C01812=1216.851,306.923,-68.303,-176.403,7.071,148.270
C01813=1216.855,306.675,-68.273,-176.405,7.069,148.270
C01814=1216.859,306.427,-68.243,-176.408,7.066,148.270
C01815=1216.864,306.178,-68.213,-176.410,7.063,148.270
C01816=1216.868,305.930,-68.183,-176.413,7.060,148.270
C01817=1216.872,305.682,-68.154,-176.415,7.058,148.270
C01818=1216.876,305.434,-68.124,-176.417,7.056,148.270
C01819=1216.881,305.186,-68.095,-176.420,7.053,148.270
C01820=1216.885,304.938,-68.064,-176.422,7.051,148.270
C01821=1216.889,304.690,-68.035,-176.424,7.048,148.270
C01822=1216.894,304.442,-68.006,-176.427,7.045,148.270
C01823=1216.898,304.193,-67.976,-176.429,7.042,148.270
C01824=1216.903,303.945,-67.946,-176.431,7.040,148.270
C01825=1216.907,303.697,-67.916,-176.434,7.038,148.270
C01826=1216.911,303.449,-67.886,-176.436,7.035,148.270
C01827=1216.915,303.201,-67.857,-176.438,7.033,148.270
C01828=1216.919,302.952,-67.827,-176.441,7.030,148.270
C01829=1216.924,302.704,-67.797,-176.443,7.028,148.270
C01830=1216.928,302.456,-67.768,-176.446,7.024,148.270
C01831=1216.932,302.207,-67.739,-176.448,7.022,148.270
C01832=1216.936,301.960,-67.708,-176.451,7.019,148.270
C01833=1216.940,301.711,-67.679,-176.453,7.017,148.270
C01834=1216.945,301.463,-67.649,-176.455,7.015,148.270
C01835=1216.950,301.215,-67.619,-176.457,7.012,148.271
C01836=1216.954,300.966,-67.590,-176.460,7.010,148.271
C01837=1216.958,300.718,-67.561,-176.463,7.007,148.271
C01838=1216.963,300.470,-67.531,-176.465,7.005,148.271
C01839=1216.967,300.222,-67.502,-176.468,7.002,148.271
C01840=1216.971,299.974,-67.473,-176.470,6.999,148.271
C01841=1216.975,299.726,-67.443,-176.472,6.997,148.271
C01842=1216.979,299.477,-67.414,-176.474,6.994,148.271
C01843=1216.984,299.229,-67.384,-176.477,6.992,148.271
C01844=1216.988,298.981,-67.355,-176.479,6.989,148.271
C01845=1216.992,298.733,-67.325,-176.481,6.987,148.271
C01846=1216.996,298.484,-67.296,-176.484,6.985,148.271
C01847=1217.001,298.237,-67.267,-176.487,6.982,148.271
C01848=1217.005,297.988,-67.238,-176.489,6.980,148.271
C01849=1217.010,297.740,-67.209,-176.491,6.976,148.271
C01850=1217.014,297.491,-67.179,-176.493,6.974,148.272
C01851=1217.018,297.243,-67.150,-176.496,6.971,148.272
C01852=1217.022,296.995,-67.120,-176.498,6.969,148.272
C01853=1217.026,296.747,-67.091,-176.500,6.967,148.272
C01854=1217.031,296.499,-67.062,-176.504,6.964,148.272
C01855=1217.036,296.250,-67.033,-176.506,6.962,148.272
C01856=1217.040,296.002,-67.003,-176.508,6.959,148.272
C01857=1217.044,295.754,-66.974,-176.510,6.957,148.272
C01858=1217.048,295.505,-66.945,-176.513,6.954,148.272
C01859=1217.053,295.258,-66.915,-176.515,6.951,148.272
C01860=1217.057,295.009,-66.887,-176.518,6.950,148.272
C01861=1217.062,294.761,-66.857,-176.521,6.946,148.272
C01862=1217.066,294.512,-66.828,-176.523,6.944,148.272
C01863=1217.070,294.264,-66.798,-176.525,6.942,148.273
C01864=1217.075,294.016,-66.770,-176.527,6.939,148.273
C01865=1217.079,293.768,-66.741,-176.530,6.937,148.273
C01866=1217.083,293.520,-66.712,-176.533,6.934,148.273
C01867=1217.087,293.271,-66.683,-176.535,6.932,148.273
C01868=1217.091,293.022,-66.653,-176.537,6.930,148.273
C01869=1217.096,292.775,-66.624,-176.540,6.927,148.273
C01870=1217.101,292.526,-66.596,-176.542,6.924,148.273
C01871=1217.105,292.278,-66.566,-176.544,6.923,148.273
C01872=1217.109,292.029,-66.537,-176.547,6.920,148.273
C01873=1217.113,291.782,-66.509,-176.549,6.917,148.273
C01874=1217.118,291.533,-66.479,-176.552,6.914,148.273
C01875=1217.122,291.284,-66.451,-176.554,6.912,148.274
C01876=1217.126,291.036,-66.421,-176.557,6.910,148.274
C01877=1217.131,290.789,-66.392,-176.559,6.907,148.274
C01878=1217.135,290.540,-66.364,-176.561,6.905,148.274
C01879=1217.139,290.292,-66.335,-176.564,6.902,148.274
C01880=1217.144,290.044,-66.306,-176.567,6.900,148.274
C01881=1217.148,289.795,-66.277,-176.569,6.898,148.274
C01882=1217.153,289.521,-66.245,-176.571,6.895,148.274
C01883=1217.158,289.247,-66.214,-176.575,6.892,148.275
C01884=1217.162,288.973,-66.181,-176.577,6.890,148.275
C01885=1217.167,288.698,-66.150,-176.579,6.887,148.275
C01886=1217.172,288.450,-66.121,-176.582,6.884,148.275
C01887=1217.176,288.202,-66.092,-176.585,6.882,148.275
C01888=1217.180,287.953,-66.064,-176.587,6.880,148.275
C01889=1217.184,287.705,-66.034,-176.589,6.877,148.275
C01890=1217.189,287.457,-66.006,-176.592,6.875,148.275
C01891=1217.193,287.208,-65.978,-176.594,6.873,148.275
C01892=1217.197,286.960,-65.948,-176.597,6.869,148.275
C01893=1217.202,286.712,-65.920,-176.599,6.868,148.276
C01894=1217.206,286.463,-65.892,-176.602,6.865,148.276
C01895=1217.210,286.215,-65.862,-176.604,6.862,148.276
C01896=1217.215,285.967,-65.834,-176.606,6.860,148.276
C01897=1217.219,285.718,-65.806,-176.609,6.857,148.276
C01898=1217.223,285.470,-65.776,-176.612,6.855,148.276
C01899=1217.228,285.222,-65.748,-176.614,6.853,148.276
C01900=1217.232,284.973,-65.720,-176.617,6.850,148.276
C01901=1217.237,284.726,-65.691,-176.619,6.848,148.276
C01902=1217.241,284.477,-65.662,-176.621,6.846,148.277
C01903=1217.245,284.228,-65.634,-176.624,6.843,148.277
C01904=1217.250,283.980,-65.605,-176.626,6.841,148.277
C01905=1217.254,283.732,-65.576,-176.629,6.839,148.277
C01906=1217.259,283.484,-65.548,-176.632,6.836,148.277
C01907=1217.263,283.235,-65.520,-176.634,6.834,148.277
C01908=1217.267,282.986,-65.491,-176.636,6.832,148.277
C01909=1217.271,282.739,-65.463,-176.639,6.829,148.278
C01910=1217.276,282.490,-65.434,-176.641,6.827,148.278
C01911=1217.280,282.242,-65.406,-176.643,6.825,148.278
C01912=1217.284,281.994,-65.377,-176.646,6.822,148.278
C01913=1217.290,281.745,-65.349,-176.649,6.820,148.278
C01914=1217.293,281.497,-65.321,-176.651,6.817,148.278
C01915=1217.298,281.249,-65.293,-176.654,6.815,148.278
C01916=1217.302,281.000,-65.264,-176.656,6.812,148.278
C01917=1217.307,280.751,-65.236,-176.658,6.810,148.278
C01918=1217.311,280.504,-65.207,-176.661,6.808,148.279
C01919=1217.314,280.255,-65.179,-176.663,6.805,148.279
C01920=1217.319,280.007,-65.151,-176.666,6.803,148.279
C01921=1217.323,279.759,-65.123,-176.669,6.800,148.279
C01922=1217.328,279.510,-65.094,-176.671,6.798,148.279
C01923=1217.332,279.262,-65.066,-176.673,6.796,148.279
C01924=1217.337,279.014,-65.038,-176.676,6.794,148.280
C01925=1217.341,278.765,-65.010,-176.678,6.791,148.280
C01926=1217.346,278.517,-64.981,-176.681,6.789,148.280
C01927=1217.350,278.268,-64.953,-176.683,6.787,148.280
C01928=1217.354,278.020,-64.925,-176.686,6.784,148.280
C01929=1217.359,277.772,-64.897,-176.688,6.782,148.280
C01930=1217.363,277.524,-64.869,-176.690,6.780,148.280
C01931=1217.368,277.274,-64.841,-176.694,6.777,148.281
C01932=1217.372,277.026,-64.813,-176.696,6.775,148.281
C01933=1217.376,276.778,-64.785,-176.698,6.773,148.281
C01934=1217.381,276.530,-64.756,-176.701,6.770,148.281
C01935=1217.385,276.281,-64.728,-176.703,6.768,148.281
C01936=1217.389,276.033,-64.700,-176.706,6.766,148.281
C01937=1217.394,275.785,-64.672,-176.708,6.764,148.281
C01938=1217.398,275.536,-64.644,-176.710,6.761,148.281
C01939=1217.403,275.288,-64.617,-176.713,6.759,148.282
C01940=1217.407,275.039,-64.588,-176.715,6.757,148.282
C01941=1217.411,274.791,-64.560,-176.718,6.754,148.282
C01942=1217.415,274.542,-64.532,-176.720,6.752,148.282
C01943=1217.420,274.294,-64.504,-176.723,6.750,148.282
C01944=1217.424,274.045,-64.476,-176.725,6.748,148.282
C01945=1217.429,273.797,-64.449,-176.728,6.745,148.283
C01946=1217.433,273.549,-64.421,-176.731,6.743,148.283
C01947=1217.437,273.300,-64.392,-176.733,6.741,148.283
C01948=1217.442,273.052,-64.365,-176.736,6.738,148.283
C01949=1217.446,272.803,-64.337,-176.738,6.736,148.283
C01950=1217.450,272.555,-64.309,-176.741,6.734,148.283
C01951=1217.455,272.307,-64.281,-176.743,6.732,148.284
C01952=1217.459,272.058,-64.253,-176.746,6.729,148.284
C01953=1217.464,271.810,-64.226,-176.748,6.727,148.284
C01954=1217.468,271.562,-64.198,-176.751,6.725,148.284
C01955=1217.472,271.313,-64.170,-176.753,6.723,148.284
C01956=1217.477,271.065,-64.142,-176.756,6.720,148.285
C01957=1217.481,270.816,-64.115,-176.758,6.718,148.285
C01958=1217.486,270.568,-64.087,-176.760,6.715,148.285
C01959=1217.490,270.320,-64.059,-176.763,6.714,148.285
C01960=1217.494,270.071,-64.032,-176.765,6.711,148.285
C01961=1217.499,269.823,-64.003,-176.768,6.709,148.285
C01962=1217.504,269.574,-63.976,-176.770,6.706,148.285
C01963=1217.508,269.326,-63.948,-176.773,6.704,148.286
C01964=1217.512,269.078,-63.920,-176.775,6.702,148.286
C01965=1217.517,268.829,-63.893,-176.778,6.700,148.286
C01966=1217.520,268.581,-63.865,-176.780,6.698,148.286
C01967=1217.525,268.332,-63.838,-176.783,6.695,148.286
C01968=1217.529,268.084,-63.810,-176.785,6.693,148.286
C01969=1217.535,267.835,-63.783,-176.788,6.691,148.287
C01970=1217.538,267.587,-63.754,-176.790,6.689,148.287
C01971=1217.543,267.338,-63.727,-176.793,6.687,148.287
C01972=1217.548,267.090,-63.700,-176.795,6.684,148.287
C01973=1217.551,266.841,-63.672,-176.798,6.682,148.287
C01974=1217.556,266.593,-63.645,-176.800,6.680,148.287
C01975=1217.560,266.345,-63.617,-176.803,6.678,148.288
C01976=1217.565,266.096,-63.590,-176.806,6.675,148.288
C01977=1217.569,265.848,-63.562,-176.808,6.673,148.288
C01978=1217.574,265.599,-63.535,-176.810,6.671,148.288
C01979=1217.578,265.351,-63.508,-176.813,6.669,148.289
C01980=1217.583,265.103,-63.480,-176.816,6.666,148.289
C01981=1217.587,264.854,-63.453,-176.818,6.664,148.289
C01982=1217.591,264.605,-63.426,-176.821,6.662,148.289
C01983=1217.596,264.357,-63.398,-176.823,6.660,148.289
C01984=1217.600,264.109,-63.371,-176.825,6.658,148.290
C01985=1217.604,263.860,-63.343,-176.828,6.655,148.290
C01986=1217.610,263.587,-63.313,-176.831,6.653,148.290
C01987=1217.614,263.315,-63.283,-176.834,6.650,148.290
C01988=1217.619,263.042,-63.253,-176.836,6.648,148.290
C01989=1217.624,262.770,-63.223,-176.839,6.645,148.290
C01990=1217.629,262.521,-63.196,-176.842,6.643,148.291
C01991=1217.633,262.272,-63.169,-176.844,6.641,148.291
C01992=1217.637,262.024,-63.142,-176.847,6.639,148.291
C01993=1217.642,261.776,-63.114,-176.849,6.636,148.291
C01994=1217.646,261.527,-63.087,-176.852,6.634,148.291
C01995=1217.651,261.279,-63.060,-176.854,6.632,148.292
C01996=1217.655,261.030,-63.033,-176.857,6.630,148.292
C01997=1217.659,260.781,-63.006,-176.859,6.629,148.292
C01998=1217.664,260.533,-62.979,-176.862,6.625,148.292
C01999=1217.668,260.285,-62.951,-176.865,6.624,148.293
C02000=1217.673,260.037,-62.924,-176.867,6.621,148.293
C02001=1217.677,259.788,-62.897,-176.869,6.620,148.293
C02002=1217.681,259.539,-62.870,-176.871,6.617,148.293
C02003=1217.686,259.290,-62.843,-176.875,6.615,148.293
C02004=1217.690,259.042,-62.816,-176.877,6.613,148.294
C02005=1217.695,258.794,-62.789,-176.879,6.611,148.294
C02006=1217.699,258.545,-62.762,-176.882,6.609,148.294
C02007=1217.704,258.297,-62.735,-176.884,6.606,148.294
C02008=1217.708,258.048,-62.708,-176.887,6.605,148.294
C02009=1217.712,257.799,-62.681,-176.890,6.602,148.295
C02010=1217.716,257.551,-62.654,-176.892,6.600,148.295
C02011=1217.721,257.302,-62.627,-176.895,6.598,148.295
C02012=1217.726,257.054,-62.600,-176.897,6.596,148.295
C02013=1217.730,256.805,-62.573,-176.899,6.594,148.295
C02014=1217.734,256.557,-62.546,-176.903,6.591,148.296
C02015=1217.739,256.309,-62.519,-176.905,6.589,148.296
C02016=1217.744,256.060,-62.492,-176.907,6.587,148.296
C02017=1217.748,255.812,-62.466,-176.909,6.585,148.296
C02018=1217.752,255.563,-62.439,-176.912,6.583,148.296
C02019=1217.757,255.315,-62.412,-176.915,6.581,148.297
C02020=1217.762,255.066,-62.385,-176.917,6.579,148.297
C02021=1217.765,254.818,-62.358,-176.920,6.576,148.297
C02022=1217.770,254.569,-62.331,-176.923,6.574,148.297
C02023=1217.774,254.320,-62.304,-176.925,6.572,148.297
C02024=1217.778,254.072,-62.278,-176.927,6.570,148.298
C02025=1217.783,253.823,-62.251,-176.929,6.568,148.298
C02026=1217.788,253.575,-62.224,-176.932,6.566,148.298
C02027=1217.792,253.327,-62.197,-176.935,6.563,148.298
C02028=1217.796,253.078,-62.170,-176.937,6.561,148.299
C02029=1217.801,252.829,-62.144,-176.940,6.559,148.299
C02030=1217.805,252.581,-62.117,-176.943,6.558,148.299
C02031=1217.810,252.332,-62.090,-176.945,6.555,148.299
C02032=1217.815,252.084,-62.063,-176.947,6.553,148.300
C02033=1217.819,251.835,-62.038,-176.950,6.552,148.300
C02034=1217.823,251.587,-62.010,-176.953,6.549,148.300
C02035=1217.827,251.338,-61.984,-176.955,6.547,148.300
C02036=1217.832,251.090,-61.957,-176.958,6.545,148.300
C02037=1217.837,250.841,-61.931,-176.960,6.543,148.301
C02038=1217.841,250.593,-61.904,-176.963,6.541,148.301
C02039=1217.845,250.344,-61.877,-176.965,6.539,148.301
C02040=1217.850,250.095,-61.851,-176.967,6.537,148.301
C02041=1217.854,249.847,-61.824,-176.970,6.535,148.302
C02042=1217.858,249.599,-61.798,-176.973,6.532,148.302
C02043=1217.863,249.349,-61.771,-176.975,6.530,148.302
C02044=1217.867,249.101,-61.745,-176.978,6.528,148.302
C02045=1217.872,248.853,-61.718,-176.981,6.526,148.303
C02046=1217.876,248.604,-61.692,-176.983,6.524,148.303
C02047=1217.881,248.355,-61.665,-176.985,6.522,148.303
C02048=1217.885,248.107,-61.639,-176.988,6.520,148.303
C02049=1217.890,247.859,-61.613,-176.990,6.518,148.303
C02050=1217.894,247.610,-61.587,-176.993,6.515,148.304
C02051=1217.899,247.362,-61.560,-176.996,6.514,148.304
C02052=1217.903,247.113,-61.533,-176.998,6.511,148.304
C02053=1217.908,246.864,-61.507,-177.001,6.509,148.304
C02054=1217.912,246.616,-61.481,-177.003,6.508,148.305
C02055=1217.917,246.367,-61.454,-177.005,6.505,148.305
C02056=1217.921,246.119,-61.428,-177.008,6.504,148.305
C02057=1217.926,245.870,-61.401,-177.011,6.502,148.305
C02058=1217.930,245.621,-61.376,-177.013,6.500,148.306
C02059=1217.935,245.372,-61.349,-177.015,6.498,148.306
C02060=1217.939,245.124,-61.323,-177.019,6.495,148.306
C02061=1217.943,244.876,-61.297,-177.021,6.493,148.306
C02062=1217.948,244.627,-61.270,-177.023,6.491,148.306
C02063=1217.952,244.379,-61.244,-177.026,6.489,148.307
C02064=1217.956,244.130,-61.218,-177.029,6.487,148.307
C02065=1217.961,243.881,-61.192,-177.031,6.485,148.307
C02066=1217.965,243.633,-61.165,-177.033,6.483,148.307
C02067=1217.970,243.384,-61.139,-177.036,6.481,148.308
C02068=1217.975,243.136,-61.113,-177.039,6.479,148.308
C02069=1217.979,242.887,-61.087,-177.041,6.477,148.308
C02070=1217.984,242.638,-61.061,-177.043,6.475,148.309
C02071=1217.988,242.390,-61.034,-177.046,6.473,148.309
C02072=1217.992,242.141,-61.009,-177.049,6.471,148.309
C02073=1217.997,241.892,-60.982,-177.051,6.469,148.309
C02074=1218.002,241.644,-60.957,-177.054,6.467,148.310
C02075=1218.006,241.396,-60.930,-177.056,6.465,148.310
C02076=1218.010,241.147,-60.905,-177.059,6.463,148.310
C02077=1218.015,240.898,-60.878,-177.061,6.461,148.310
C02078=1218.019,240.649,-60.853,-177.064,6.459,148.311
C02079=1218.024,240.402,-60.826,-177.066,6.457,148.311
C02080=1218.029,240.152,-60.800,-177.069,6.455,148.311
C02081=1218.033,239.904,-60.774,-177.071,6.453,148.311
C02082=1218.037,239.655,-60.749,-177.074,6.451,148.312
C02083=1218.041,239.407,-60.722,-177.076,6.449,148.312
C02084=1218.047,239.158,-60.696,-177.079,6.447,148.312
C02085=1218.051,238.909,-60.670,-177.082,6.444,148.312
C02086=1218.055,238.661,-60.645,-177.084,6.443,148.313
C02087=1218.059,238.412,-60.619,-177.087,6.441,148.313
C02088=1218.064,238.164,-60.594,-177.090,6.439,148.313
C02089=1218.069,237.915,-60.567,-177.092,6.437,148.313
C02090=1218.074,237.643,-60.538,-177.094,6.435,148.314
C02091=1218.079,237.372,-60.511,-177.097,6.433,148.314
C02092=1218.083,237.101,-60.482,-177.100,6.430,148.314
C02093=1218.088,236.829,-60.454,-177.103,6.428,148.315
C02094=1218.093,236.581,-60.429,-177.105,6.426,148.315
C02095=1218.097,236.332,-60.403,-177.108,6.425,148.315
C02096=1218.101,236.083,-60.377,-177.111,6.423,148.316
C02097=1218.107,235.835,-60.351,-177.113,6.421,148.316
C02098=1218.111,235.586,-60.325,-177.115,6.419,148.316
C02099=1218.115,235.337,-60.300,-177.118,6.417,148.316
C02100=1218.119,235.088,-60.274,-177.121,6.415,148.317
C02101=1218.124,234.840,-60.248,-177.123,6.413,148.317
C02102=1218.128,234.592,-60.223,-177.125,6.411,148.317
C02103=1218.133,234.343,-60.197,-177.128,6.409,148.317
C02104=1218.138,234.095,-60.172,-177.131,6.406,148.318
C02105=1218.142,233.846,-60.146,-177.134,6.404,148.318
C02106=1218.146,233.597,-60.120,-177.137,6.403,148.318
C02107=1218.152,233.349,-60.094,-177.139,6.400,148.318
C02108=1218.156,233.100,-60.068,-177.141,6.399,148.319
C02109=1218.160,232.851,-60.043,-177.144,6.397,148.319
C02110=1218.165,232.602,-60.018,-177.147,6.395,148.319
C02111=1218.169,232.353,-59.992,-177.149,6.393,148.320
C02112=1218.174,232.105,-59.966,-177.151,6.391,148.320
C02113=1218.178,231.857,-59.941,-177.154,6.389,148.320
C02114=1218.183,231.608,-59.915,-177.157,6.387,148.320
C02115=1218.187,231.359,-59.890,-177.159,6.385,148.321
C02116=1218.192,231.110,-59.865,-177.162,6.383,148.321
C02117=1218.196,230.861,-59.839,-177.164,6.382,148.321
C02118=1218.201,230.613,-59.814,-177.167,6.379,148.321
C02119=1218.205,230.364,-59.788,-177.169,6.377,148.322
C02120=1218.209,230.116,-59.762,-177.172,6.376,148.322
C02121=1218.215,229.867,-59.738,-177.174,6.374,148.322
C02122=1218.219,229.618,-59.712,-177.177,6.372,148.323
C02123=1218.223,229.369,-59.686,-177.180,6.370,148.323
C02124=1218.227,229.122,-59.661,-177.182,6.368,148.323
C02125=1218.232,228.872,-59.636,-177.185,6.366,148.323
C02126=1218.236,228.624,-59.611,-177.187,6.364,148.324
C02127=1218.241,228.375,-59.585,-177.190,6.362,148.324
C02128=1218.246,228.127,-59.560,-177.192,6.360,148.324
C02129=1218.250,227.878,-59.535,-177.195,6.359,148.325
C02130=1218.254,227.629,-59.509,-177.197,6.356,148.325
C02131=1218.259,227.380,-59.484,-177.200,6.355,148.325
C02132=1218.264,227.131,-59.459,-177.202,6.353,148.326
C02133=1218.268,226.883,-59.433,-177.205,6.351,148.326
C02134=1218.272,226.634,-59.409,-177.208,6.349,148.326
C02135=1218.277,226.386,-59.383,-177.210,6.347,148.326
C02136=1218.281,226.137,-59.358,-177.213,6.345,148.327
C02137=1218.286,225.889,-59.333,-177.215,6.343,148.327
C02138=1218.291,225.640,-59.307,-177.218,6.341,148.327
C02139=1218.295,225.390,-59.282,-177.220,6.339,148.328
C02140=1218.300,225.142,-59.257,-177.223,6.338,148.328
C02141=1218.304,224.893,-59.232,-177.226,6.336,148.328
C02142=1218.309,224.645,-59.207,-177.228,6.334,148.329
C02143=1218.313,224.396,-59.182,-177.231,6.332,148.329
C02144=1218.318,224.147,-59.156,-177.234,6.330,148.329
C02145=1218.323,223.898,-59.131,-177.236,6.328,148.329
C02146=1218.327,223.650,-59.107,-177.238,6.326,148.330
C02147=1218.331,223.401,-59.082,-177.241,6.324,148.330
C02148=1218.336,223.153,-59.056,-177.244,6.322,148.330
C02149=1218.341,222.903,-59.031,-177.246,6.320,148.331
C02150=1218.345,222.655,-59.006,-177.249,6.319,148.331
C02151=1218.349,222.406,-58.981,-177.251,6.317,148.331
C02152=1218.354,222.158,-58.956,-177.254,6.315,148.332
C02153=1218.359,221.909,-58.931,-177.257,6.313,148.332
C02154=1218.363,221.660,-58.907,-177.259,6.311,148.332
C02155=1218.368,221.412,-58.881,-177.261,6.309,148.332
C02156=1218.372,221.163,-58.856,-177.264,6.307,148.333
C02157=1218.376,220.915,-58.832,-177.266,6.306,148.333
C02158=1218.381,220.665,-58.807,-177.269,6.304,148.333
C02159=1218.386,220.417,-58.782,-177.271,6.302,148.334
C02160=1218.389,220.168,-58.757,-177.274,6.301,148.334
C02161=1218.395,219.919,-58.732,-177.277,6.299,148.334
C02162=1218.400,219.671,-58.707,-177.279,6.297,148.335
C02163=1218.403,219.422,-58.682,-177.282,6.295,148.335
C02164=1218.408,219.173,-58.658,-177.285,6.293,148.335
C02165=1218.413,218.924,-58.633,-177.287,6.291,148.336
C02166=1218.417,218.676,-58.609,-177.290,6.290,148.336
C02167=1218.422,218.427,-58.583,-177.292,6.287,148.336
C02168=1218.426,218.178,-58.559,-177.295,6.285,148.336
C02169=1218.431,217.930,-58.534,-177.297,6.284,148.337
C02170=1218.436,217.680,-58.509,-177.300,6.282,148.337
C02171=1218.440,217.432,-58.484,-177.303,6.280,148.337
C02172=1218.445,217.184,-58.460,-177.305,6.278,148.338
C02173=1218.449,216.935,-58.435,-177.308,6.276,148.338
C02174=1218.454,216.686,-58.410,-177.310,6.274,148.338
C02175=1218.458,216.436,-58.385,-177.313,6.273,148.339
C02176=1218.463,216.188,-58.361,-177.316,6.271,148.339
C02177=1218.467,215.940,-58.336,-177.318,6.269,148.339
C02178=1218.471,215.691,-58.311,-177.321,6.267,148.340
C02179=1218.476,215.442,-58.287,-177.324,6.265,148.340
C02180=1218.481,215.194,-58.263,-177.326,6.263,148.340
C02181=1218.485,214.944,-58.238,-177.328,6.262,148.341
C02182=1218.490,214.696,-58.214,-177.331,6.260,148.341
C02183=1218.495,214.447,-58.189,-177.334,6.259,148.341
C02184=1218.499,214.198,-58.165,-177.336,6.257,148.342
C02185=1218.504,213.949,-58.140,-177.339,6.255,148.342
C02186=1218.508,213.701,-58.116,-177.342,6.253,148.342
C02187=1218.513,213.451,-58.091,-177.344,6.251,148.343
C02188=1218.517,213.204,-58.066,-177.346,6.249,148.343
C02189=1218.522,212.955,-58.041,-177.349,6.247,148.343
C02190=1218.526,212.706,-58.017,-177.352,6.245,148.344
C02191=1218.531,212.457,-57.992,-177.354,6.243,148.344
C02192=1218.535,212.209,-57.968,-177.357,6.242,148.344
C02193=1218.540,211.960,-57.945,-177.359,6.240,148.345
C02194=1218.544,211.689,-57.918,-177.362,6.238,148.345
C02195=1218.550,211.419,-57.891,-177.365,6.236,148.345
C02196=1218.555,211.148,-57.864,-177.368,6.235,148.346
C02197=1218.560,210.878,-57.838,-177.371,6.233,148.346
C02198=1218.564,210.629,-57.814,-177.373,6.231,148.346
C02199=1218.569,210.380,-57.789,-177.376,6.229,148.347
C02200=1218.574,210.131,-57.765,-177.378,6.227,148.347
C02201=1218.578,209.883,-57.741,-177.381,6.225,148.347
C02202=1218.582,209.634,-57.716,-177.384,6.223,148.348
C02203=1218.587,209.385,-57.692,-177.386,6.222,148.348
C02204=1218.591,209.137,-57.668,-177.389,6.220,148.348
C02205=1218.596,208.888,-57.643,-177.392,6.218,148.349
C02206=1218.601,208.639,-57.620,-177.394,6.216,148.349
C02207=1218.605,208.390,-57.595,-177.396,6.215,148.350
C02208=1218.610,208.141,-57.571,-177.399,6.213,148.350
C02209=1218.614,207.893,-57.547,-177.402,6.211,148.350
C02210=1218.619,207.644,-57.523,-177.404,6.210,148.351
C02211=1218.624,207.394,-57.498,-177.407,6.208,148.351
C02212=1218.628,207.146,-57.474,-177.410,6.206,148.351
C02213=1218.632,206.898,-57.450,-177.412,6.204,148.352
C02214=1218.638,206.649,-57.425,-177.415,6.202,148.352
C02215=1218.642,206.400,-57.402,-177.417,6.200,148.352
C02216=1218.647,206.151,-57.378,-177.420,6.199,148.353
C02217=1218.650,205.902,-57.354,-177.422,6.197,148.353
C02218=1218.656,205.653,-57.330,-177.425,6.196,148.353
C02219=1218.660,205.404,-57.305,-177.427,6.194,148.354
C02220=1218.665,205.156,-57.281,-177.430,6.192,148.354
C02221=1218.669,204.908,-57.257,-177.433,6.190,148.354
C02222=1218.675,204.658,-57.233,-177.435,6.188,148.355
C02223=1218.678,204.409,-57.209,-177.438,6.186,148.355
C02224=1218.683,204.160,-57.186,-177.441,6.185,148.355
C02225=1218.687,203.912,-57.162,-177.443,6.184,148.356
C02226=1218.692,203.663,-57.137,-177.445,6.182,148.356
C02227=1218.697,203.414,-57.114,-177.448,6.180,148.356
C02228=1218.702,203.166,-57.089,-177.451,6.178,148.357
C02229=1218.706,202.917,-57.066,-177.453,6.176,148.357
C02230=1218.710,202.667,-57.042,-177.456,6.174,148.357
C02231=1218.715,202.419,-57.018,-177.459,6.172,148.358
C02232=1218.719,202.170,-56.994,-177.461,6.171,148.358
C02233=1218.724,201.922,-56.970,-177.463,6.170,148.358
C02234=1218.729,201.672,-56.946,-177.466,6.168,148.359
C02235=1218.733,201.424,-56.922,-177.469,6.166,148.359
C02236=1218.738,201.175,-56.899,-177.472,6.164,148.360
C02237=1218.743,200.926,-56.875,-177.474,6.163,148.360
C02238=1218.747,200.677,-56.851,-177.477,6.161,148.360
C02239=1218.752,200.429,-56.827,-177.479,6.160,148.361
C02240=1218.756,200.179,-56.803,-177.482,6.158,148.361
C02241=1218.760,199.931,-56.779,-177.484,6.156,148.361
C02242=1218.765,199.682,-56.756,-177.487,6.154,148.362
C02243=1218.769,199.433,-56.732,-177.490,6.152,148.362
C02244=1218.775,199.184,-56.708,-177.492,6.151,148.362
C02245=1218.779,198.935,-56.685,-177.494,6.150,148.363
C02246=1218.784,198.687,-56.661,-177.497,6.148,148.363
C02247=1218.788,198.438,-56.637,-177.500,6.146,148.363
C02248=1218.793,198.189,-56.613,-177.502,6.144,148.364
C02249=1218.798,197.940,-56.590,-177.505,6.142,148.364
C02250=1218.802,197.691,-56.566,-177.508,6.140,148.365
C02251=1218.807,197.443,-56.542,-177.510,6.139,148.365
C02252=1218.811,197.194,-56.519,-177.512,6.137,148.365
C02253=1218.816,196.945,-56.496,-177.515,6.136,148.366
C02254=1218.820,196.696,-56.472,-177.518,6.134,148.366
C02255=1218.825,196.447,-56.448,-177.521,6.132,148.366
C02256=1218.830,196.198,-56.425,-177.523,6.130,148.367
C02257=1218.835,195.949,-56.401,-177.525,6.129,148.367
C02258=1218.839,195.701,-56.377,-177.528,6.128,148.368
C02259=1218.844,195.452,-56.354,-177.531,6.126,148.368
C02260=1218.848,195.203,-56.331,-177.533,6.124,148.368
C02261=1218.853,194.954,-56.307,-177.536,6.122,148.369
C02262=1218.857,194.705,-56.284,-177.538,6.121,148.369
C02263=1218.861,194.456,-56.260,-177.541,6.119,148.369
C02264=1218.866,194.207,-56.237,-177.543,6.117,148.370
C02265=1218.871,193.958,-56.214,-177.547,6.116,148.370
C02266=1218.875,193.710,-56.190,-177.549,6.114,148.371
C02267=1218.880,193.461,-56.166,-177.551,6.113,148.371
C02268=1218.885,193.212,-56.143,-177.554,6.111,148.371
C02269=1218.889,192.963,-56.120,-177.557,6.109,148.372
C02270=1218.894,192.714,-56.096,-177.559,6.108,148.372
C02271=1218.899,192.465,-56.073,-177.562,6.106,148.372
C02272=1218.903,192.216,-56.050,-177.564,6.105,148.373
C02273=1218.908,191.968,-56.026,-177.567,6.103,148.373
C02274=1218.912,191.719,-56.003,-177.569,6.101,148.373
C02275=1218.917,191.470,-55.980,-177.572,6.100,148.374
C02276=1218.922,191.221,-55.956,-177.575,6.098,148.374
C02277=1218.926,190.972,-55.933,-177.577,6.097,148.375
C02278=1218.931,190.723,-55.910,-177.580,6.095,148.375
C02279=1218.935,190.474,-55.887,-177.582,6.093,148.375
C02280=1218.940,190.225,-55.864,-177.585,6.091,148.376
C02281=1218.944,189.976,-55.840,-177.587,6.090,148.376
C02282=1218.949,189.727,-55.817,-177.590,6.088,148.376
C02283=1218.954,189.479,-55.794,-177.592,6.087,148.377
C02284=1218.958,189.230,-55.771,-177.596,6.085,148.377
C02285=1218.963,188.981,-55.748,-177.598,6.083,148.378
C02286=1218.968,188.732,-55.724,-177.600,6.082,148.378
C02287=1218.973,188.483,-55.701,-177.603,6.080,148.378
C02288=1218.977,188.234,-55.678,-177.606,6.078,148.379
C02289=1218.981,187.985,-55.655,-177.608,6.077,148.379
C02290=1218.986,187.736,-55.631,-177.610,6.076,148.380
C02291=1218.991,187.488,-55.608,-177.613,6.074,148.380
C02292=1218.995,187.239,-55.586,-177.616,6.072,148.380
C02293=1219.000,186.990,-55.562,-177.619,6.070,148.381
C02294=1219.005,186.741,-55.539,-177.621,6.069,148.381
C02295=1219.010,186.492,-55.516,-177.624,6.068,148.382
C02296=1219.014,186.243,-55.494,-177.626,6.066,148.382
C02297=1219.019,185.995,-55.471,-177.629,6.064,148.382
C02298=1219.024,185.725,-55.446,-177.632,6.062,148.383
C02299=1219.029,185.455,-55.421,-177.635,6.061,148.383
C02300=1219.034,185.186,-55.396,-177.637,6.059,148.384
C02301=1219.038,184.915,-55.371,-177.640,6.057,148.384
C02302=1219.043,184.667,-55.348,-177.642,6.056,148.384
C02303=1219.048,184.418,-55.325,-177.645,6.055,148.385
C02304=1219.052,184.169,-55.302,-177.648,6.053,148.385
C02305=1219.057,183.920,-55.279,-177.650,6.051,148.386
C02306=1219.062,183.671,-55.257,-177.653,6.050,148.386
C02307=1219.066,183.423,-55.234,-177.655,6.048,148.386
C02308=1219.071,183.174,-55.210,-177.658,6.047,148.387
C02309=1219.075,182.925,-55.188,-177.661,6.045,148.387
C02310=1219.080,182.675,-55.165,-177.663,6.044,148.388
C02311=1219.085,182.427,-55.142,-177.666,6.042,148.388
C02312=1219.089,182.178,-55.119,-177.668,6.040,148.388
C02313=1219.094,181.929,-55.096,-177.670,6.039,148.389
C02314=1219.098,181.680,-55.074,-177.674,6.038,148.389
C02315=1219.103,181.432,-55.051,-177.676,6.036,148.390
C02316=1219.107,181.183,-55.028,-177.679,6.034,148.390
C02317=1219.112,180.933,-55.005,-177.681,6.033,148.390
C02318=1219.117,180.684,-54.982,-177.684,6.031,148.391
C02319=1219.122,180.435,-54.960,-177.687,6.030,148.391
C02320=1219.127,180.186,-54.937,-177.689,6.029,148.392
C02321=1219.131,179.938,-54.914,-177.692,6.027,148.392
C02322=1219.136,179.689,-54.892,-177.694,6.025,148.392
C02323=1219.140,179.440,-54.869,-177.697,6.023,148.393
C02324=1219.145,179.190,-54.847,-177.699,6.022,148.393
C02325=1219.149,178.942,-54.824,-177.702,6.021,148.394
C02326=1219.155,178.693,-54.801,-177.705,6.019,148.394
C02327=1219.159,178.444,-54.779,-177.707,6.018,148.394
C02328=1219.163,178.195,-54.755,-177.709,6.016,148.395
C02329=1219.168,177.946,-54.734,-177.712,6.014,148.395
C02330=1219.172,177.698,-54.711,-177.715,6.013,148.396
C02331=1219.177,177.448,-54.688,-177.717,6.012,148.396
C02332=1219.182,177.200,-54.666,-177.720,6.010,148.396
C02333=1219.187,176.950,-54.643,-177.723,6.008,148.397
C02334=1219.191,176.702,-54.621,-177.725,6.007,148.397
C02335=1219.196,176.453,-54.598,-177.728,6.005,148.398
C02336=1219.200,176.204,-54.576,-177.731,6.004,148.398
C02337=1219.205,175.955,-54.553,-177.733,6.003,148.399
C02338=1219.210,175.706,-54.530,-177.735,6.001,148.399
C02339=1219.214,175.457,-54.508,-177.738,5.999,148.399
C02340=1219.219,175.207,-54.486,-177.741,5.998,148.400
C02341=1219.224,174.959,-54.463,-177.743,5.997,148.400
C02342=1219.228,174.710,-54.441,-177.746,5.995,148.401
C02343=1219.233,174.462,-54.418,-177.748,5.994,148.401
C02344=1219.238,174.212,-54.396,-177.751,5.992,148.401
C02345=1219.242,173.963,-54.374,-177.754,5.990,148.402
C02346=1219.247,173.715,-54.351,-177.756,5.989,148.402
C02347=1219.252,173.465,-54.329,-177.758,5.988,148.403
C02348=1219.257,173.216,-54.307,-177.761,5.986,148.403
C02349=1219.261,172.967,-54.284,-177.764,5.985,148.404
C02350=1219.265,172.718,-54.262,-177.766,5.983,148.404
C02351=1219.270,172.470,-54.240,-177.769,5.981,148.404
C02352=1219.275,172.220,-54.217,-177.771,5.980,148.405
C02353=1219.280,171.972,-54.195,-177.774,5.979,148.405
C02354=1219.284,171.722,-54.173,-177.777,5.977,148.406
C02355=1219.289,171.473,-54.151,-177.779,5.976,148.406
C02356=1219.294,171.225,-54.128,-177.782,5.974,148.406
C02357=1219.298,170.975,-54.106,-177.784,5.972,148.407
C02358=1219.303,170.727,-54.085,-177.787,5.972,148.407
C02359=1219.308,170.477,-54.062,-177.790,5.970,148.408
C02360=1219.312,170.229,-54.040,-177.792,5.968,148.408
C02361=1219.317,169.980,-54.017,-177.794,5.967,148.409
C02362=1219.321,169.731,-53.996,-177.798,5.966,148.409
C02363=1219.326,169.482,-53.973,-177.800,5.964,148.409
C02364=1219.331,169.233,-53.951,-177.802,5.963,148.410
C02365=1219.336,168.984,-53.929,-177.805,5.961,148.410
C02366=1219.340,168.736,-53.907,-177.808,5.960,148.411
C02367=1219.345,168.486,-53.884,-177.810,5.959,148.411
C02368=1219.349,168.237,-53.862,-177.813,5.957,148.412
C02369=1219.354,167.988,-53.841,-177.815,5.956,148.412
C02370=1219.359,167.739,-53.819,-177.818,5.954,148.413
C02371=1219.363,167.490,-53.797,-177.821,5.952,148.413
C02372=1219.368,167.240,-53.774,-177.823,5.951,148.413
C02373=1219.373,166.992,-53.753,-177.825,5.950,148.414
C02374=1219.378,166.742,-53.731,-177.829,5.948,148.414
C02375=1219.382,166.494,-53.709,-177.831,5.947,148.415
C02376=1219.387,166.246,-53.686,-177.833,5.945,148.415
C02377=1219.391,165.996,-53.664,-177.836,5.944,148.415
C02378=1219.396,165.748,-53.643,-177.839,5.943,148.416
C02379=1219.400,165.498,-53.621,-177.841,5.941,148.416
C02380=1219.406,165.249,-53.598,-177.843,5.940,148.417
C02381=1219.410,165.000,-53.576,-177.846,5.938,148.417
C02382=1219.415,164.751,-53.555,-177.849,5.937,148.418
C02383=1219.419,164.502,-53.533,-177.851,5.936,148.418
C02384=1219.424,164.253,-53.511,-177.854,5.934,148.418
C02385=1219.429,164.004,-53.489,-177.857,5.933,148.419
C02386=1219.433,163.755,-53.467,-177.859,5.932,148.419
C02387=1219.438,163.505,-53.446,-177.862,5.930,148.420
C02388=1219.443,163.257,-53.424,-177.864,5.929,148.420
C02389=1219.448,163.008,-53.403,-177.867,5.927,148.421
C02390=1219.452,162.759,-53.380,-177.869,5.926,148.421
C02391=1219.457,162.510,-53.359,-177.872,5.924,148.422
C02392=1219.461,162.261,-53.337,-177.875,5.923,148.422
C02393=1219.466,162.012,-53.315,-177.877,5.922,148.422
C02394=1219.471,161.764,-53.293,-177.880,5.920,148.423
C02395=1219.475,161.514,-53.271,-177.882,5.919,148.423
C02396=1219.480,161.265,-53.250,-177.885,5.918,148.424
C02397=1219.485,161.016,-53.228,-177.888,5.916,148.424
C02398=1219.489,160.767,-53.207,-177.890,5.915,148.425
C02399=1219.494,160.518,-53.185,-177.893,5.913,148.425
C02400=1219.499,160.269,-53.163,-177.895,5.912,148.426
C02401=1219.503,160.020,-53.141,-177.898,5.911,148.426
C02402=1219.509,159.751,-53.118,-177.901,5.909,148.427
C02403=1219.514,159.482,-53.094,-177.904,5.907,148.427
C02404=1219.519,159.213,-53.071,-177.906,5.907,148.428
C02405=1219.524,158.944,-53.048,-177.909,5.905,148.428
C02406=1219.529,158.694,-53.026,-177.912,5.903,148.429
C02407=1219.534,158.445,-53.005,-177.914,5.902,148.429
C02408=1219.538,158.197,-52.984,-177.917,5.901,148.429
C02409=1219.542,157.948,-52.962,-177.919,5.900,148.430
C02410=1219.547,157.698,-52.941,-177.922,5.898,148.430
C02411=1219.552,157.450,-52.919,-177.925,5.896,148.431
C02412=1219.557,157.200,-52.897,-177.927,5.895,148.431
C02413=1219.561,156.952,-52.875,-177.930,5.894,148.432
C02414=1219.567,156.702,-52.854,-177.932,5.893,148.432
C02415=1219.571,156.453,-52.832,-177.935,5.891,148.432
C02416=1219.576,156.204,-52.810,-177.937,5.890,148.433
C02417=1219.580,155.956,-52.790,-177.940,5.889,148.433
C02418=1219.585,155.707,-52.768,-177.942,5.888,148.434
C02419=1219.590,155.457,-52.747,-177.945,5.886,148.434
C02420=1219.594,155.208,-52.725,-177.948,5.884,148.435
C02421=1219.599,154.960,-52.704,-177.950,5.883,148.435
C02422=1219.604,154.710,-52.682,-177.953,5.882,148.436
C02423=1219.608,154.461,-52.661,-177.955,5.881,148.436
C02424=1219.613,154.212,-52.640,-177.958,5.879,148.436
C02425=1219.618,153.963,-52.619,-177.960,5.878,148.437
C02426=1219.623,153.713,-52.597,-177.963,5.877,148.437
C02427=1219.628,153.465,-52.576,-177.965,5.876,148.438
C02428=1219.633,153.216,-52.555,-177.968,5.874,148.438
C02429=1219.637,152.967,-52.534,-177.971,5.872,148.439
C02430=1219.641,152.717,-52.512,-177.973,5.871,148.439
C02431=1219.646,152.469,-52.491,-177.976,5.870,148.440
C02432=1219.651,152.219,-52.470,-177.978,5.869,148.440
C02433=1219.656,151.971,-52.448,-177.981,5.867,148.441
C02434=1219.660,151.721,-52.427,-177.984,5.866,148.441
C02435=1219.665,151.472,-52.405,-177.986,5.865,148.442
C02436=1219.670,151.223,-52.384,-177.989,5.864,148.442
C02437=1219.674,150.975,-52.363,-177.992,5.862,148.443
C02438=1219.680,150.726,-52.342,-177.994,5.861,148.443
C02439=1219.684,150.476,-52.320,-177.997,5.860,148.444
C02440=1219.688,150.227,-52.300,-177.999,5.859,148.444
C02441=1219.693,149.978,-52.279,-178.002,5.857,148.444
C02442=1219.698,149.729,-52.257,-178.004,5.856,148.445
C02443=1219.703,149.480,-52.236,-178.007,5.854,148.445
C02444=1219.707,149.231,-52.215,-178.009,5.853,148.446
C02445=1219.712,148.982,-52.194,-178.012,5.852,148.446
C02446=1219.717,148.733,-52.173,-178.014,5.851,148.447
C02447=1219.721,148.484,-52.152,-178.017,5.850,148.447
C02448=1219.727,148.235,-52.131,-178.020,5.849,148.448
C02449=1219.730,147.985,-52.110,-178.022,5.847,148.448
C02450=1219.735,147.737,-52.089,-178.025,5.845,148.449
C02451=1219.740,147.487,-52.068,-178.027,5.844,148.449
C02452=1219.745,147.239,-52.047,-178.030,5.843,148.450
C02453=1219.750,146.989,-52.026,-178.033,5.842,148.450
C02454=1219.755,146.741,-52.005,-178.035,5.840,148.451
C02455=1219.759,146.492,-51.984,-178.038,5.839,148.451
C02456=1219.764,146.242,-51.963,-178.041,5.838,148.452
C02457=1219.768,145.993,-51.942,-178.043,5.837,148.452
C02458=1219.773,145.744,-51.921,-178.046,5.835,148.453
C02459=1219.778,145.495,-51.900,-178.048,5.834,148.453
C02460=1219.783,145.246,-51.879,-178.051,5.834,148.454
C02461=1219.788,144.997,-51.858,-178.053,5.832,148.454
C02462=1219.792,144.748,-51.837,-178.055,5.831,148.454
C02463=1219.797,144.499,-51.816,-178.059,5.829,148.455
C02464=1219.801,144.249,-51.796,-178.061,5.828,148.455
C02465=1219.806,144.000,-51.775,-178.063,5.827,148.456
C02466=1219.811,143.751,-51.754,-178.066,5.826,148.456
C02467=1219.816,143.502,-51.733,-178.069,5.824,148.457
C02468=1219.820,143.253,-51.713,-178.071,5.823,148.457
C02469=1219.825,143.004,-51.691,-178.074,5.822,148.458
C02470=1219.830,142.755,-51.671,-178.077,5.821,148.458
C02471=1219.835,142.506,-51.650,-178.079,5.819,148.459
C02472=1219.839,142.257,-51.630,-178.081,5.818,148.459
C02473=1219.845,142.008,-51.609,-178.084,5.817,148.460
C02474=1219.849,141.759,-51.588,-178.087,5.816,148.460
C02475=1219.854,141.510,-51.567,-178.090,5.814,148.461
C02476=1219.858,141.260,-51.547,-178.092,5.813,148.461
C02477=1219.863,141.011,-51.526,-178.095,5.812,148.462
C02478=1219.868,140.762,-51.505,-178.097,5.811,148.462
C02479=1219.873,140.513,-51.484,-178.100,5.809,148.463
C02480=1219.877,140.264,-51.464,-178.102,5.809,148.463
C02481=1219.882,140.014,-51.443,-178.104,5.808,148.464
C02482=1219.887,139.765,-51.423,-178.107,5.806,148.464
C02483=1219.891,139.516,-51.402,-178.110,5.805,148.465
C02484=1219.896,139.267,-51.381,-178.112,5.803,148.465
C02485=1219.901,139.018,-51.361,-178.115,5.803,148.466
C02486=1219.906,138.769,-51.340,-178.118,5.801,148.466
C02487=1219.910,138.520,-51.320,-178.120,5.800,148.467
C02488=1219.915,138.271,-51.299,-178.123,5.798,148.467
C02489=1219.920,138.022,-51.278,-178.125,5.797,148.467
C02490=1219.925,137.773,-51.258,-178.128,5.796,148.468
C02491=1219.929,137.524,-51.237,-178.130,5.795,148.468
C02492=1219.934,137.275,-51.216,-178.133,5.794,148.469
C02493=1219.939,137.026,-51.196,-178.136,5.793,148.469
C02494=1219.944,136.777,-51.175,-178.138,5.792,148.470
C02495=1219.948,136.527,-51.155,-178.141,5.790,148.470
C02496=1219.953,136.278,-51.135,-178.144,5.790,148.471
C02497=1219.958,136.029,-51.114,-178.146,5.788,148.471
C02498=1219.963,135.780,-51.094,-178.148,5.787,148.472
C02499=1219.967,135.531,-51.073,-178.151,5.785,148.472
C02500=1219.971,135.282,-51.053,-178.154,5.784,148.473
C02501=1219.977,135.032,-51.033,-178.156,5.784,148.473
C02502=1219.982,134.784,-51.013,-178.159,5.782,148.474
C02503=1219.986,134.535,-50.992,-178.161,5.781,148.474
C02504=1219.992,134.286,-50.971,-178.164,5.779,148.475
C02505=1219.996,134.037,-50.951,-178.167,5.779,148.475
C02506=1220.002,133.768,-50.929,-178.169,5.777,148.476
C02507=1220.006,133.499,-50.907,-178.172,5.776,148.477
C02508=1220.011,133.230,-50.886,-178.175,5.775,148.477
C02509=1220.017,132.962,-50.863,-178.178,5.773,148.477
C02510=1220.021,132.712,-50.843,-178.180,5.773,148.478
C02511=1220.026,132.463,-50.823,-178.183,5.772,148.479
C02512=1220.030,132.214,-50.803,-178.186,5.770,148.479
C02513=1220.035,131.965,-50.782,-178.188,5.769,148.480
C02514=1220.041,131.716,-50.762,-178.191,5.768,148.480
C02515=1220.045,131.467,-50.742,-178.193,5.767,148.481
C02516=1220.050,131.218,-50.722,-178.195,5.766,148.481
C02517=1220.054,130.969,-50.702,-178.198,5.764,148.482
C02518=1220.059,130.720,-50.682,-178.201,5.763,148.482
C02519=1220.064,130.470,-50.661,-178.204,5.762,148.483
C02520=1220.069,130.221,-50.641,-178.206,5.761,148.483
C02521=1220.073,129.972,-50.621,-178.208,5.760,148.484
C02522=1220.079,129.723,-50.601,-178.211,5.758,148.484
C02523=1220.083,129.474,-50.581,-178.214,5.758,148.485
C02524=1220.087,129.225,-50.561,-178.216,5.756,148.485
C02525=1220.093,128.975,-50.540,-178.219,5.755,148.486
C02526=1220.097,128.726,-50.520,-178.221,5.754,148.486
C02527=1220.102,128.477,-50.500,-178.224,5.753,148.487
C02528=1220.107,128.228,-50.480,-178.226,5.752,148.487
C02529=1220.112,127.979,-50.461,-178.230,5.751,148.488
C02530=1220.116,127.730,-50.440,-178.232,5.750,148.488
C02531=1220.121,127.480,-50.421,-178.234,5.749,148.489
C02532=1220.125,127.231,-50.400,-178.237,5.747,148.489
C02533=1220.130,126.982,-50.381,-178.240,5.747,148.490
C02534=1220.135,126.733,-50.360,-178.242,5.746,148.490
C02535=1220.141,126.484,-50.340,-178.245,5.744,148.491
C02536=1220.145,126.235,-50.320,-178.247,5.743,148.491
C02537=1220.150,125.985,-50.300,-178.250,5.742,148.492
C02538=1220.154,125.736,-50.280,-178.252,5.741,148.492
C02539=1220.159,125.487,-50.260,-178.255,5.740,148.493
C02540=1220.164,125.238,-50.240,-178.258,5.738,148.493
C02541=1220.169,124.989,-50.221,-178.260,5.738,148.494
C02542=1220.173,124.740,-50.200,-178.262,5.737,148.494
C02543=1220.178,124.490,-50.181,-178.265,5.735,148.495
C02544=1220.183,124.241,-50.161,-178.268,5.734,148.495
C02545=1220.188,123.992,-50.141,-178.271,5.733,148.496
C02546=1220.193,123.743,-50.121,-178.273,5.732,148.496
C02547=1220.197,123.494,-50.101,-178.275,5.731,148.497
C02548=1220.202,123.245,-50.082,-178.278,5.730,148.497
C02549=1220.207,122.996,-50.062,-178.281,5.729,148.498
C02550=1220.212,122.747,-50.042,-178.283,5.728,148.498
C02551=1220.216,122.497,-50.022,-178.286,5.727,148.499
C02552=1220.222,122.248,-50.003,-178.288,5.726,148.499
C02553=1220.226,121.999,-49.982,-178.291,5.725,148.500
C02554=1220.231,121.750,-49.963,-178.293,5.723,148.500
C02555=1220.236,121.500,-49.943,-178.296,5.723,148.501
C02556=1220.241,121.252,-49.923,-178.298,5.722,148.502
C02557=1220.245,121.002,-49.903,-178.301,5.720,148.502
C02558=1220.250,120.753,-49.884,-178.304,5.720,148.503
C02559=1220.254,120.503,-49.865,-178.307,5.718,148.503
C02560=1220.259,120.255,-49.845,-178.309,5.717,148.504
C02561=1220.264,120.006,-49.825,-178.311,5.716,148.504
C02562=1220.269,119.756,-49.805,-178.315,5.715,148.505
C02563=1220.274,119.507,-49.786,-178.317,5.714,148.505
C02564=1220.279,119.258,-49.766,-178.319,5.713,148.506
C02565=1220.283,119.009,-49.746,-178.322,5.711,148.506
C02566=1220.288,118.760,-49.727,-178.325,5.711,148.507
C02567=1220.293,118.510,-49.707,-178.327,5.710,148.507
C02568=1220.297,118.261,-49.688,-178.330,5.708,148.508
C02569=1220.303,118.012,-49.669,-178.332,5.707,148.508
C02570=1220.307,117.763,-49.648,-178.335,5.707,148.509
C02571=1220.312,117.514,-49.629,-178.337,5.705,148.509
C02572=1220.317,117.265,-49.609,-178.340,5.704,148.510
C02573=1220.322,117.015,-49.590,-178.342,5.704,148.511
C02574=1220.327,116.766,-49.570,-178.345,5.702,148.511
C02575=1220.331,116.517,-49.551,-178.348,5.701,148.512
C02576=1220.336,116.267,-49.532,-178.350,5.700,148.512
C02577=1220.341,116.018,-49.512,-178.353,5.700,148.513
C02578=1220.346,115.769,-49.493,-178.355,5.698,148.513
C02579=1220.350,115.520,-49.472,-178.358,5.697,148.514
C02580=1220.355,115.272,-49.454,-178.360,5.696,148.514
C02581=1220.360,115.022,-49.434,-178.363,5.695,148.515
C02582=1220.365,114.772,-49.414,-178.366,5.694,148.516
C02583=1220.370,114.524,-49.395,-178.368,5.693,148.516
C02584=1220.374,114.274,-49.376,-178.371,5.692,148.517
C02585=1220.379,114.025,-49.357,-178.373,5.691,148.517
C02586=1220.384,113.776,-49.337,-178.376,5.690,148.518
C02587=1220.389,113.526,-49.317,-178.378,5.689,148.518
C02588=1220.393,113.278,-49.299,-178.381,5.688,148.519
C02589=1220.398,113.028,-49.279,-178.384,5.687,148.519
C02590=1220.403,112.779,-49.260,-178.386,5.686,148.520
C02591=1220.408,112.530,-49.240,-178.389,5.685,148.520
C02592=1220.412,112.280,-49.221,-178.391,5.684,148.521
C02593=1220.418,112.032,-49.202,-178.394,5.683,148.521
C02594=1220.422,111.782,-49.182,-178.396,5.682,148.522
C02595=1220.427,111.533,-49.164,-178.399,5.681,148.522
C02596=1220.432,111.283,-49.144,-178.402,5.680,148.523
C02597=1220.437,111.034,-49.125,-178.404,5.679,148.523
C02598=1220.441,110.785,-49.106,-178.407,5.678,148.524
C02599=1220.447,110.536,-49.087,-178.409,5.677,148.525
C02600=1220.451,110.287,-49.067,-178.412,5.676,148.525
C02601=1220.455,110.037,-49.048,-178.414,5.675,148.526
C02602=1220.461,109.789,-49.029,-178.417,5.674,148.526
C02603=1220.465,109.539,-49.009,-178.420,5.673,148.527
C02604=1220.470,109.290,-48.991,-178.422,5.672,148.527
C02605=1220.475,109.040,-48.972,-178.425,5.671,148.528
C02606=1220.480,108.791,-48.952,-178.427,5.670,148.528
C02607=1220.484,108.542,-48.933,-178.430,5.669,148.529
C02608=1220.490,108.293,-48.914,-178.433,5.668,148.530
C02609=1220.494,108.043,-48.896,-178.435,5.667,148.530
C02610=1220.500,107.775,-48.875,-178.438,5.666,148.531
C02611=1220.505,107.507,-48.854,-178.441,5.665,148.531
C02612=1220.510,107.238,-48.834,-178.443,5.664,148.532
C02613=1220.515,106.970,-48.813,-178.446,5.663,148.532
C02614=1220.520,106.721,-48.794,-178.449,5.662,148.533
C02615=1220.525,106.471,-48.774,-178.451,5.661,148.534
C02616=1220.530,106.222,-48.756,-178.453,5.660,148.534
C02617=1220.534,105.973,-48.737,-178.457,5.659,148.535
C02618=1220.539,105.724,-48.718,-178.459,5.658,148.535
C02619=1220.545,105.475,-48.699,-178.461,5.657,148.536
C02620=1220.549,105.225,-48.680,-178.464,5.657,148.536
C02621=1220.554,104.977,-48.661,-178.467,5.655,148.537
C02622=1220.559,104.726,-48.642,-178.469,5.654,148.537
C02623=1220.564,104.478,-48.623,-178.471,5.654,148.538
C02624=1220.568,104.228,-48.604,-178.474,5.653,148.538
C02625=1220.573,103.979,-48.586,-178.477,5.651,148.539
C02626=1220.578,103.729,-48.566,-178.479,5.651,148.539
C02627=1220.583,103.481,-48.547,-178.482,5.650,148.540
C02628=1220.587,103.232,-48.529,-178.484,5.649,148.541
C02629=1220.592,102.982,-48.510,-178.487,5.648,148.541
C02630=1220.597,102.733,-48.492,-178.490,5.647,148.542
C02631=1220.602,102.483,-48.472,-178.492,5.646,148.542
C02632=1220.606,102.235,-48.453,-178.495,5.645,148.543
C02633=1220.611,101.985,-48.435,-178.498,5.644,148.544
C02634=1220.616,101.736,-48.416,-178.500,5.643,148.544
C02635=1220.622,101.487,-48.397,-178.502,5.642,148.545
C02636=1220.626,101.237,-48.378,-178.505,5.642,148.545
C02637=1220.631,100.988,-48.360,-178.508,5.640,148.546
C02638=1220.635,100.739,-48.341,-178.510,5.639,148.546
C02639=1220.640,100.489,-48.323,-178.512,5.638,148.547
C02640=1220.646,100.241,-48.303,-178.515,5.638,148.547
C02641=1220.650,99.991,-48.284,-178.518,5.636,148.548
C02642=1220.655,99.742,-48.266,-178.520,5.636,148.548
C02643=1220.660,99.493,-48.248,-178.523,5.635,148.549
C02644=1220.664,99.243,-48.229,-178.526,5.634,148.550
C02645=1220.670,98.994,-48.210,-178.528,5.633,148.550
C02646=1220.674,98.745,-48.191,-178.531,5.632,148.551
C02647=1220.679,98.496,-48.173,-178.534,5.631,148.551
C02648=1220.684,98.247,-48.154,-178.536,5.630,148.552
C02649=1220.688,97.997,-48.135,-178.538,5.630,148.552
C02650=1220.693,97.748,-48.117,-178.541,5.628,148.553
C02651=1220.699,97.499,-48.098,-178.544,5.627,148.554
C02652=1220.703,97.249,-48.080,-178.546,5.627,148.554
C02653=1220.708,97.000,-48.061,-178.548,5.626,148.555
C02654=1220.713,96.751,-48.042,-178.551,5.625,148.555
C02655=1220.718,96.502,-48.024,-178.554,5.624,148.556
C02656=1220.722,96.252,-48.005,-178.556,5.623,148.556
C02657=1220.728,96.003,-47.987,-178.559,5.622,148.557
C02658=1220.732,95.754,-47.968,-178.562,5.622,148.558
C02659=1220.737,95.504,-47.950,-178.564,5.621,148.558
C02660=1220.742,95.255,-47.931,-178.567,5.619,148.559
C02661=1220.747,95.006,-47.913,-178.569,5.619,148.559
C02662=1220.751,94.757,-47.894,-178.572,5.618,148.560
C02663=1220.756,94.507,-47.876,-178.574,5.617,148.560
C02664=1220.762,94.258,-47.857,-178.577,5.617,148.561
C02665=1220.766,94.009,-47.839,-178.580,5.615,148.561
C02666=1220.771,93.759,-47.821,-178.582,5.614,148.562
C02667=1220.776,93.510,-47.803,-178.585,5.614,148.563
C02668=1220.781,93.261,-47.783,-178.587,5.613,148.563
C02669=1220.785,93.012,-47.765,-178.590,5.612,148.564
C02670=1220.790,92.762,-47.747,-178.593,5.611,148.564
C02671=1220.795,92.513,-47.729,-178.595,5.610,148.565
C02672=1220.800,92.265,-47.710,-178.597,5.609,148.566
C02673=1220.805,92.014,-47.691,-178.600,5.609,148.566
C02674=1220.810,91.765,-47.673,-178.602,5.608,148.567
C02675=1220.815,91.516,-47.655,-178.605,5.607,148.567
C02676=1220.820,91.267,-47.637,-178.608,5.606,148.568
C02677=1220.824,91.018,-47.619,-178.610,5.605,148.568
C02678=1220.829,90.768,-47.600,-178.613,5.604,148.569
C02679=1220.834,90.519,-47.582,-178.615,5.603,148.570
C02680=1220.839,90.270,-47.564,-178.618,5.602,148.570
C02681=1220.844,90.021,-47.546,-178.621,5.601,148.571
C02682=1220.848,89.771,-47.528,-178.623,5.600,148.571
C02683=1220.853,89.522,-47.510,-178.625,5.600,148.572
C02684=1220.858,89.272,-47.492,-178.628,5.599,148.572
C02685=1220.863,89.024,-47.473,-178.631,5.598,148.573
C02686=1220.868,88.774,-47.454,-178.633,5.598,148.574
C02687=1220.873,88.524,-47.436,-178.636,5.596,148.574
C02688=1220.878,88.275,-47.418,-178.639,5.595,148.575
C02689=1220.883,88.026,-47.400,-178.641,5.595,148.575
C02690=1220.887,87.777,-47.382,-178.643,5.594,148.576
C02691=1220.892,87.528,-47.364,-178.646,5.593,148.577
C02692=1220.897,87.279,-47.346,-178.649,5.593,148.577
C02693=1220.902,87.029,-47.328,-178.651,5.592,148.578
C02694=1220.906,86.780,-47.310,-178.654,5.590,148.578
C02695=1220.911,86.530,-47.292,-178.657,5.590,148.579
C02696=1220.916,86.281,-47.274,-178.659,5.589,148.580
C02697=1220.921,86.032,-47.256,-178.661,5.588,148.580
C02698=1220.926,85.783,-47.238,-178.664,5.588,148.581
C02699=1220.931,85.533,-47.219,-178.667,5.587,148.581
C02700=1220.936,85.283,-47.201,-178.669,5.585,148.582
C02701=1220.941,85.034,-47.183,-178.672,5.585,148.582
C02702=1220.946,84.785,-47.165,-178.675,5.584,148.583
C02703=1220.951,84.536,-47.147,-178.677,5.583,148.583
C02704=1220.956,84.287,-47.129,-178.679,5.583,148.584
C02705=1220.961,84.038,-47.111,-178.682,5.582,148.585
C02706=1220.966,83.788,-47.093,-178.685,5.581,148.585
C02707=1220.970,83.539,-47.075,-178.687,5.580,148.586
C02708=1220.975,83.289,-47.057,-178.690,5.579,148.586
C02709=1220.980,83.040,-47.039,-178.693,5.578,148.587
C02710=1220.985,82.790,-47.021,-178.695,5.577,148.588
C02711=1220.989,82.542,-47.004,-178.697,5.577,148.588
C02712=1220.994,82.292,-46.986,-178.700,5.576,148.589
C02713=1220.999,82.043,-46.968,-178.703,5.576,148.590
C02714=1221.004,81.775,-46.949,-178.705,5.574,148.590
C02715=1221.009,81.506,-46.930,-178.708,5.573,148.591
C02716=1221.015,81.237,-46.910,-178.710,5.573,148.591
C02717=1221.020,80.969,-46.891,-178.713,5.572,148.592
C02718=1221.024,80.720,-46.873,-178.716,5.571,148.593
C02719=1221.030,80.471,-46.856,-178.719,5.570,148.593
C02720=1221.035,80.221,-46.838,-178.721,5.569,148.594
C02721=1221.039,79.972,-46.820,-178.724,5.569,148.594
C02722=1221.044,79.723,-46.802,-178.726,5.568,148.595
C02723=1221.050,79.473,-46.785,-178.729,5.568,148.596
C02724=1221.055,79.224,-46.767,-178.731,5.567,148.596
C02725=1221.059,78.975,-46.749,-178.734,5.566,148.597
C02726=1221.064,78.726,-46.731,-178.737,5.565,148.597
C02727=1221.069,78.476,-46.714,-178.740,5.564,148.598
C02728=1221.074,78.227,-46.696,-178.742,5.563,148.598
C02729=1221.079,77.978,-46.678,-178.744,5.562,148.599
C02730=1221.084,77.729,-46.660,-178.747,5.562,148.600
C02731=1221.089,77.479,-46.643,-178.750,5.561,148.600
C02732=1221.094,77.230,-46.625,-178.752,5.560,148.601
C02733=1221.099,76.981,-46.607,-178.754,5.560,148.601
C02734=1221.103,76.731,-46.590,-178.757,5.559,148.602
C02735=1221.108,76.482,-46.572,-178.760,5.557,148.603
C02736=1221.113,76.233,-46.554,-178.762,5.557,148.603
C02737=1221.118,75.983,-46.537,-178.765,5.556,148.604
C02738=1221.123,75.734,-46.519,-178.768,5.556,148.605
C02739=1221.127,75.485,-46.502,-178.770,5.555,148.605
C02740=1221.132,75.235,-46.484,-178.772,5.554,148.606
C02741=1221.137,74.986,-46.466,-178.775,5.554,148.606
C02742=1221.143,74.736,-46.449,-178.778,5.553,148.607
C02743=1221.147,74.487,-46.432,-178.780,5.552,148.607
C02744=1221.152,74.238,-46.414,-178.782,5.552,148.608
C02745=1221.157,73.988,-46.397,-178.785,5.551,148.609
C02746=1221.162,73.739,-46.379,-178.788,5.550,148.609
C02747=1221.166,73.490,-46.362,-178.790,5.549,148.610
C02748=1221.171,73.240,-46.344,-178.793,5.548,148.610
C02749=1221.176,72.991,-46.327,-178.796,5.547,148.611
C02750=1221.181,72.742,-46.309,-178.798,5.547,148.612
C02751=1221.186,72.492,-46.292,-178.801,5.546,148.612
C02752=1221.191,72.243,-46.274,-178.803,5.545,148.613
C02753=1221.196,71.993,-46.257,-178.806,5.545,148.613
C02754=1221.200,71.744,-46.239,-178.808,5.544,148.614
C02755=1221.205,71.494,-46.222,-178.811,5.544,148.615
C02756=1221.210,71.245,-46.204,-178.813,5.543,148.615
C02757=1221.216,70.996,-46.187,-178.816,5.542,148.616
C02758=1221.220,70.747,-46.170,-178.818,5.542,148.617
C02759=1221.225,70.497,-46.153,-178.821,5.540,148.617
C02760=1221.230,70.248,-46.135,-178.824,5.539,148.618
C02761=1221.235,69.999,-46.118,-178.826,5.539,148.618
C02762=1221.240,69.749,-46.101,-178.829,5.538,148.619
C02763=1221.245,69.500,-46.083,-178.831,5.537,148.620
C02764=1221.249,69.250,-46.066,-178.834,5.537,148.620
C02765=1221.254,69.001,-46.048,-178.836,5.536,148.621
C02766=1221.259,68.752,-46.031,-178.839,5.535,148.621
C02767=1221.265,68.503,-46.014,-178.841,5.535,148.622
C02768=1221.270,68.253,-45.997,-178.844,5.534,148.623
C02769=1221.274,68.004,-45.980,-178.846,5.533,148.623
C02770=1221.279,67.755,-45.962,-178.849,5.533,148.624
C02771=1221.283,67.505,-45.945,-178.851,5.532,148.624
C02772=1221.289,67.255,-45.928,-178.854,5.532,148.625
C02773=1221.294,67.006,-45.910,-178.856,5.531,148.626
C02774=1221.299,66.758,-45.894,-178.859,5.530,148.626
C02775=1221.304,66.508,-45.876,-178.862,5.529,148.627
C02776=1221.308,66.258,-45.860,-178.865,5.528,148.628
C02777=1221.313,66.009,-45.842,-178.867,5.528,148.628
C02778=1221.318,65.760,-45.825,-178.869,5.527,148.629
C02779=1221.323,65.510,-45.808,-178.872,5.526,148.629
C02780=1221.327,65.261,-45.790,-178.875,5.525,148.630
C02781=1221.333,65.012,-45.774,-178.877,5.525,148.631
C02782=1221.338,64.762,-45.756,-178.880,5.524,148.631
C02783=1221.343,64.513,-45.740,-178.882,5.523,148.632
C02784=1221.348,64.263,-45.722,-178.885,5.523,148.632
C02785=1221.352,64.014,-45.705,-178.887,5.522,148.633
C02786=1221.358,63.765,-45.688,-178.890,5.522,148.634
C02787=1221.362,63.515,-45.671,-178.893,5.521,148.634
C02788=1221.368,63.266,-45.654,-178.895,5.520,148.635
C02789=1221.372,63.017,-45.637,-178.897,5.520,148.635
C02790=1221.377,62.767,-45.619,-178.900,5.519,148.636
C02791=1221.382,62.518,-45.603,-178.903,5.518,148.637
C02792=1221.387,62.268,-45.586,-178.905,5.518,148.637
C02793=1221.392,62.019,-45.569,-178.907,5.517,148.638
C02794=1221.396,61.769,-45.553,-178.910,5.516,148.639
C02795=1221.402,61.521,-45.535,-178.913,5.516,148.639
C02796=1221.406,61.271,-45.518,-178.915,5.515,148.640
C02797=1221.411,61.022,-45.501,-178.918,5.515,148.641
C02798=1221.416,60.772,-45.484,-178.920,5.514,148.641
C02799=1221.422,60.523,-45.467,-178.923,5.513,148.642
C02800=1221.426,60.273,-45.451,-178.925,5.513,148.642
C02801=1221.431,60.024,-45.433,-178.928,5.512,148.643
C02802=1221.436,59.774,-45.417,-178.931,5.511,148.644
C02803=1221.441,59.525,-45.401,-178.933,5.511,148.644
C02804=1221.446,59.276,-45.383,-178.935,5.510,148.645
C02805=1221.450,59.027,-45.366,-178.938,5.509,148.645
C02806=1221.456,58.777,-45.349,-178.941,5.509,148.646
C02807=1221.461,58.528,-45.332,-178.943,5.508,148.647
C02808=1221.465,58.279,-45.316,-178.945,5.507,148.647
C02809=1221.470,58.029,-45.298,-178.948,5.507,148.648
C02810=1221.475,57.780,-45.282,-178.951,5.506,148.649
C02811=1221.480,57.531,-45.265,-178.954,5.505,148.649
C02812=1221.485,57.281,-45.248,-178.957,5.504,148.650
C02813=1221.490,57.031,-45.231,-178.959,5.504,148.651
C02814=1221.495,56.783,-45.215,-178.961,5.503,148.651
C02815=1221.500,56.533,-45.198,-178.964,5.502,148.652
C02816=1221.504,56.283,-45.181,-178.967,5.502,148.652
C02817=1221.509,56.035,-45.165,-178.969,5.501,148.653
C02818=1221.515,55.765,-45.147,-178.972,5.500,148.654
C02819=1221.520,55.497,-45.129,-178.975,5.500,148.654
C02820=1221.526,55.228,-45.111,-178.977,5.499,148.655
C02821=1221.531,54.960,-45.093,-178.980,5.499,148.656
C02822=1221.536,54.710,-45.077,-178.982,5.498,148.656
C02823=1221.540,54.461,-45.060,-178.985,5.498,148.657
C02824=1221.546,54.212,-45.043,-178.987,5.497,148.657
C02825=1221.551,53.962,-45.027,-178.990,5.496,148.658
C02826=1221.556,53.713,-45.010,-178.993,5.496,148.659
C02827=1221.561,53.464,-44.993,-178.995,5.495,148.659
C02828=1221.565,53.214,-44.976,-178.998,5.494,148.660
C02829=1221.570,52.965,-44.960,-179.000,5.494,148.661
C02830=1221.575,52.715,-44.944,-179.003,5.493,148.661
C02831=1221.580,52.466,-44.927,-179.005,5.492,148.662
C02832=1221.586,52.217,-44.911,-179.008,5.492,148.663
C02833=1221.590,51.967,-44.894,-179.010,5.491,148.663
C02834=1221.595,51.718,-44.877,-179.013,5.491,148.664
C02835=1221.600,51.469,-44.861,-179.016,5.490,148.665
C02836=1221.605,51.219,-44.844,-179.018,5.489,148.665
C02837=1221.610,50.970,-44.828,-179.021,5.489,148.666
C02838=1221.615,50.720,-44.811,-179.023,5.488,148.666
C02839=1221.619,50.471,-44.795,-179.026,5.488,148.667
C02840=1221.625,50.221,-44.779,-179.028,5.487,148.668
C02841=1221.630,49.972,-44.762,-179.031,5.486,148.668
C02842=1221.635,49.723,-44.746,-179.034,5.486,148.669
C02843=1221.639,49.473,-44.729,-179.036,5.485,148.669
C02844=1221.644,49.223,-44.713,-179.038,5.484,148.670
C02845=1221.649,48.974,-44.697,-179.041,5.484,148.671
C02846=1221.654,48.725,-44.680,-179.044,5.483,148.671
C02847=1221.659,48.476,-44.664,-179.046,5.483,148.672
C02848=1221.664,48.226,-44.647,-179.048,5.483,148.673
C02849=1221.669,47.977,-44.631,-179.051,5.482,148.673
C02850=1221.674,47.727,-44.615,-179.053,5.482,148.674
C02851=1221.679,47.477,-44.598,-179.056,5.481,148.675
C02852=1221.684,47.229,-44.582,-179.059,5.480,148.675
C02853=1221.689,46.979,-44.566,-179.061,5.480,148.676
C02854=1221.694,46.730,-44.550,-179.064,5.479,148.677
C02855=1221.698,46.480,-44.533,-179.066,5.479,148.677
C02856=1221.704,46.231,-44.517,-179.069,5.478,148.678
C02857=1221.709,45.981,-44.500,-179.071,5.477,148.678
C02858=1221.714,45.732,-44.484,-179.074,5.477,148.679
C02859=1221.719,45.482,-44.468,-179.076,5.476,148.680
C02860=1221.724,45.233,-44.452,-179.079,5.476,148.680
C02861=1221.728,44.983,-44.436,-179.082,5.475,148.681
C02862=1221.733,44.735,-44.419,-179.084,5.474,148.682
C02863=1221.738,44.484,-44.403,-179.087,5.474,148.682
C02864=1221.743,44.236,-44.387,-179.089,5.473,148.683
C02865=1221.748,43.986,-44.370,-179.092,5.472,148.683
C02866=1221.753,43.737,-44.355,-179.094,5.472,148.684
C02867=1221.758,43.487,-44.338,-179.097,5.471,148.685
C02868=1221.763,43.238,-44.322,-179.099,5.472,148.686
C02869=1221.768,42.988,-44.306,-179.102,5.471,148.686
C02870=1221.773,42.739,-44.290,-179.104,5.471,148.687
C02871=1221.777,42.489,-44.274,-179.107,5.470,148.687
C02872=1221.783,42.240,-44.258,-179.109,5.469,148.688
C02873=1221.787,41.991,-44.241,-179.112,5.468,148.689
C02874=1221.793,41.741,-44.226,-179.115,5.468,148.689
C02875=1221.797,41.492,-44.209,-179.117,5.467,148.690
C02876=1221.803,41.242,-44.193,-179.120,5.467,148.691
C02877=1221.807,40.992,-44.178,-179.122,5.466,148.691
C02878=1221.812,40.743,-44.161,-179.125,5.465,148.692
C02879=1221.818,40.494,-44.146,-179.127,5.465,148.692
C02880=1221.822,40.245,-44.129,-179.130,5.464,148.693
C02881=1221.828,39.995,-44.113,-179.133,5.464,148.694
C02882=1221.832,39.746,-44.097,-179.135,5.463,148.694
C02883=1221.838,39.496,-44.081,-179.137,5.463,148.695
C02884=1221.842,39.246,-44.065,-179.140,5.463,148.696
C02885=1221.847,38.997,-44.049,-179.143,5.462,148.697
C02886=1221.853,38.748,-44.033,-179.145,5.461,148.697
C02887=1221.858,38.498,-44.017,-179.147,5.461,148.698
C02888=1221.862,38.249,-44.002,-179.150,5.460,148.698
C02889=1221.867,37.999,-43.986,-179.153,5.460,148.699
C02890=1221.872,37.750,-43.970,-179.155,5.459,148.700
C02891=1221.877,37.501,-43.954,-179.158,5.459,148.700
C02892=1221.882,37.251,-43.938,-179.161,5.458,148.701
C02893=1221.887,37.002,-43.922,-179.163,5.458,148.702
C02894=1221.892,36.752,-43.906,-179.165,5.458,148.702
C02895=1221.897,36.503,-43.890,-179.167,5.457,148.703
C02896=1221.903,36.253,-43.874,-179.170,5.456,148.703
C02897=1221.906,36.004,-43.858,-179.173,5.456,148.704
C02898=1221.912,35.755,-43.843,-179.175,5.455,148.705
C02899=1221.917,35.505,-43.827,-179.178,5.455,148.706
C02900=1221.922,35.255,-43.811,-179.181,5.454,148.706
C02901=1221.927,35.006,-43.795,-179.183,5.454,148.707
C02902=1221.932,34.756,-43.779,-179.186,5.453,148.708
C02903=1221.936,34.507,-43.764,-179.188,5.453,148.708
C02904=1221.942,34.258,-43.748,-179.191,5.452,148.709
C02905=1221.946,34.008,-43.732,-179.193,5.452,148.709
C02906=1221.952,33.759,-43.716,-179.195,5.451,148.710
C02907=1221.957,33.510,-43.700,-179.198,5.451,148.711
C02908=1221.961,33.260,-43.685,-179.201,5.450,148.711
C02909=1221.966,33.010,-43.670,-179.203,5.450,148.712
C02910=1221.972,32.761,-43.654,-179.206,5.449,148.713
C02911=1221.976,32.511,-43.637,-179.209,5.449,148.713
C02912=1221.981,32.262,-43.622,-179.211,5.448,148.714
C02913=1221.986,32.013,-43.607,-179.214,5.448,148.715
C02914=1221.991,31.763,-43.591,-179.215,5.447,148.715
C02915=1221.997,31.513,-43.575,-179.218,5.447,148.716
C02916=1222.001,31.264,-43.560,-179.221,5.446,148.717
C02917=1222.006,31.014,-43.544,-179.223,5.446,148.717
C02918=1222.011,30.765,-43.528,-179.226,5.445,148.718
C02919=1222.016,30.516,-43.512,-179.229,5.445,148.719
C02920=1222.021,30.267,-43.497,-179.231,5.444,148.719
C02921=1222.026,30.017,-43.481,-179.234,5.444,148.720
C02922=1222.031,29.748,-43.464,-179.237,5.443,148.721
C02923=1222.037,29.479,-43.448,-179.239,5.443,148.721
C02924=1222.042,29.211,-43.432,-179.242,5.442,148.722
C02925=1222.048,28.943,-43.415,-179.245,5.441,148.723
C02926=1222.052,28.693,-43.399,-179.247,5.441,148.723
C02927=1222.058,28.443,-43.383,-179.249,5.441,148.724
C02928=1222.063,28.194,-43.368,-179.252,5.441,148.725
C02929=1222.068,27.945,-43.352,-179.255,5.440,148.725
C02930=1222.073,27.695,-43.337,-179.257,5.440,148.726
C02931=1222.077,27.445,-43.322,-179.260,5.439,148.727
C02932=1222.083,27.196,-43.306,-179.262,5.438,148.727
C02933=1222.087,26.947,-43.291,-179.265,5.438,148.728
C02934=1222.092,26.697,-43.275,-179.267,5.437,148.729
C02935=1222.098,26.447,-43.259,-179.269,5.437,148.729
C02936=1222.102,26.198,-43.244,-179.272,5.437,148.730
C02937=1222.108,25.949,-43.229,-179.275,5.436,148.731
C02938=1222.113,25.700,-43.213,-179.277,5.436,148.731
C02939=1222.117,25.450,-43.198,-179.280,5.435,148.732
C02940=1222.122,25.200,-43.182,-179.283,5.435,148.733
C02941=1222.127,24.951,-43.167,-179.285,5.434,148.733
C02942=1222.132,24.702,-43.152,-179.287,5.434,148.734
C02943=1222.138,24.451,-43.136,-179.290,5.434,148.735
C02944=1222.142,24.202,-43.121,-179.293,5.433,148.735
C02945=1222.148,23.953,-43.106,-179.295,5.433,148.736
C02946=1222.152,23.704,-43.091,-179.297,5.432,148.736
C02947=1222.158,23.454,-43.075,-179.300,5.431,148.737
C02948=1222.162,23.204,-43.060,-179.303,5.431,148.738
C02949=1222.167,22.955,-43.044,-179.305,5.431,148.739
C02950=1222.172,22.706,-43.029,-179.307,5.430,148.739
C02951=1222.177,22.456,-43.015,-179.310,5.430,148.740
C02952=1222.183,22.206,-42.999,-179.313,5.429,148.741
C02953=1222.187,21.957,-42.984,-179.315,5.429,148.741
C02954=1222.192,21.707,-42.968,-179.318,5.428,148.742
C02955=1222.197,21.458,-42.953,-179.320,5.429,148.743
C02956=1222.203,21.208,-42.938,-179.323,5.428,148.743
C02957=1222.207,20.959,-42.923,-179.325,5.428,148.744
C02958=1222.213,20.710,-42.908,-179.328,5.427,148.745
C02959=1222.217,20.461,-42.893,-179.330,5.426,148.745
C02960=1222.223,20.211,-42.877,-179.333,5.426,148.746
C02961=1222.227,19.961,-42.862,-179.335,5.425,148.746
C02962=1222.232,19.711,-42.847,-179.337,5.425,148.747
C02963=1222.237,19.462,-42.832,-179.340,5.425,148.748
C02964=1222.242,19.213,-42.816,-179.343,5.424,148.749
C02965=1222.247,18.963,-42.802,-179.345,5.424,148.749
C02966=1222.253,18.714,-42.786,-179.348,5.423,148.750
C02967=1222.257,18.465,-42.771,-179.351,5.423,148.751
C02968=1222.262,18.215,-42.757,-179.353,5.423,148.751
C02969=1222.267,17.965,-42.741,-179.355,5.422,148.752
C02970=1222.272,17.716,-42.726,-179.358,5.422,148.753
C02971=1222.277,17.466,-42.711,-179.361,5.421,148.753
C02972=1222.282,17.217,-42.696,-179.363,5.421,148.754
C02973=1222.288,16.967,-42.681,-179.365,5.421,148.754
C02974=1222.292,16.718,-42.666,-179.368,5.420,148.755
C02975=1222.297,16.468,-42.651,-179.370,5.420,148.756
C02976=1222.302,16.219,-42.636,-179.373,5.419,148.756
C02977=1222.307,15.969,-42.621,-179.376,5.419,148.757
C02978=1222.313,15.720,-42.606,-179.378,5.418,148.758
C02979=1222.317,15.471,-42.591,-179.380,5.418,148.759
C02980=1222.322,15.220,-42.576,-179.383,5.418,148.759
C02981=1222.327,14.971,-42.561,-179.386,5.417,148.760
C02982=1222.332,14.721,-42.546,-179.388,5.417,148.761
C02983=1222.338,14.472,-42.531,-179.391,5.416,148.761
C02984=1222.342,14.223,-42.516,-179.393,5.416,148.762
C02985=1222.347,13.973,-42.502,-179.396,5.416,148.763
C02986=1222.353,13.724,-42.486,-179.398,5.415,148.763
C02987=1222.358,13.474,-42.472,-179.401,5.415,148.764
C02988=1222.362,13.225,-42.457,-179.404,5.414,148.765
C02989=1222.368,12.975,-42.442,-179.406,5.414,148.765
C02990=1222.373,12.726,-42.427,-179.408,5.414,148.766
C02991=1222.377,12.476,-42.413,-179.410,5.413,148.766
C02992=1222.383,12.227,-42.397,-179.413,5.413,148.767
C02993=1222.388,11.977,-42.383,-179.416,5.412,148.768
C02994=1222.392,11.728,-42.368,-179.418,5.412,148.769
C02995=1222.397,11.478,-42.353,-179.420,5.412,148.769
C02996=1222.403,11.229,-42.338,-179.423,5.411,148.770
C02997=1222.408,10.979,-42.324,-179.426,5.411,148.771
C02998=1222.412,10.730,-42.309,-179.428,5.410,148.771
C02999=1222.418,10.480,-42.294,-179.431,5.410,148.772
C03000=1222.423,10.231,-42.279,-179.433,5.410,148.773
C03001=1222.428,9.981,-42.264,-179.436,5.410,148.773
C03002=1222.432,9.732,-42.249,-179.438,5.409,148.774
C03003=1222.438,9.482,-42.235,-179.441,5.409,148.775
C03004=1222.443,9.232,-42.220,-179.444,5.408,148.775
C03005=1222.448,8.983,-42.205,-179.446,5.408,148.776
C03006=1222.453,8.734,-42.191,-179.448,5.408,148.777
C03007=1222.458,8.484,-42.175,-179.451,5.407,148.777
C03008=1222.463,8.234,-42.161,-179.454,5.407,148.778
C03009=1222.468,7.985,-42.147,-179.456,5.407,148.779
C03010=1222.473,7.736,-42.132,-179.458,5.406,148.779
C03011=1222.477,7.486,-42.118,-179.461,5.406,148.780
C03012=1222.483,7.236,-42.103,-179.463,5.405,148.781
C03013=1222.488,6.987,-42.088,-179.466,5.405,148.781
C03014=1222.493,6.737,-42.073,-179.468,5.405,148.782
C03015=1222.498,6.487,-42.059,-179.471,5.404,148.783
C03016=1222.502,6.238,-42.044,-179.473,5.404,148.783
C03017=1222.508,5.988,-42.029,-179.476,5.403,148.784
C03018=1222.514,5.739,-42.015,-179.479,5.403,148.785
C03019=1222.518,5.490,-42.000,-179.481,5.403,148.785
C03020=1222.523,5.240,-41.986,-179.483,5.402,148.786
C03021=1222.528,4.991,-41.972,-179.486,5.402,148.787
C03022=1222.533,4.742,-41.957,-179.489,5.401,148.788
C03023=1222.538,4.492,-41.943,-179.491,5.402,148.788
C03024=1222.544,4.242,-41.928,-179.493,5.401,148.789
C03025=1222.548,3.992,-41.913,-179.496,5.401,148.790
C03026=1222.554,3.723,-41.898,-179.499,5.400,148.790
C03027=1222.559,3.455,-41.882,-179.501,5.400,148.791
C03028=1222.564,3.186,-41.866,-179.504,5.399,148.792
C03029=1222.570,2.917,-41.852,-179.507,5.399,148.793
C03030=1222.576,2.667,-41.837,-179.509,5.399,148.793
C03031=1222.580,2.418,-41.822,-179.512,5.399,148.794
C03032=1222.585,2.168,-41.808,-179.514,5.398,148.794
C03033=1222.590,1.919,-41.793,-179.517,5.397,148.795
C03034=1222.595,1.669,-41.779,-179.519,5.398,148.796
C03035=1222.600,1.419,-41.765,-179.521,5.397,148.796
C03036=1222.605,1.170,-41.750,-179.524,5.397,148.797
C03037=1222.610,0.921,-41.736,-179.527,5.396,148.798
C03038=1222.615,0.671,-41.722,-179.529,5.396,148.799
C03039=1222.620,0.422,-41.707,-179.531,5.396,148.799
C03040=1222.625,0.172,-41.693,-179.534,5.395,148.800
C03041=1222.630,-0.078,-41.679,-179.537,5.395,148.801
C03042=1222.635,-0.328,-41.664,-179.539,5.394,148.801
C03043=1222.640,-0.577,-41.650,-179.541,5.395,148.802
C03044=1222.645,-0.826,-41.635,-179.544,5.394,148.803
C03045=1222.650,-1.075,-41.621,-179.547,5.394,148.803
C03046=1222.655,-1.325,-41.607,-179.549,5.393,148.804
C03047=1222.660,-1.575,-41.593,-179.551,5.393,148.805
C03048=1222.665,-1.824,-41.578,-179.554,5.393,148.805
C03049=1222.671,-2.073,-41.564,-179.557,5.392,148.806
C03050=1222.676,-2.323,-41.550,-179.559,5.392,148.807
C03051=1222.680,-2.573,-41.536,-179.562,5.392,148.808
C03052=1222.685,-2.823,-41.522,-179.564,5.392,148.808
C03053=1222.690,-3.072,-41.507,-179.567,5.391,148.809
C03054=1222.695,-3.322,-41.493,-179.570,5.391,148.810
C03055=1222.701,-3.571,-41.479,-179.572,5.391,148.810
C03056=1222.706,-3.821,-41.465,-179.574,5.390,148.811
C03057=1222.711,-4.070,-41.451,-179.577,5.390,148.812
C03058=1222.716,-4.320,-41.436,-179.579,5.390,148.812
C03059=1222.721,-4.569,-41.422,-179.582,5.390,148.813
C03060=1222.726,-4.819,-41.408,-179.584,5.389,148.814
C03061=1222.731,-5.069,-41.394,-179.587,5.389,148.814
C03062=1222.736,-5.318,-41.380,-179.589,5.389,148.815
C03063=1222.741,-5.568,-41.365,-179.592,5.388,148.816
C03064=1222.747,-5.817,-41.351,-179.594,5.388,148.816
C03065=1222.752,-6.067,-41.337,-179.596,5.387,148.817
C03066=1222.757,-6.316,-41.323,-179.599,5.387,148.818
C03067=1222.761,-6.566,-41.309,-179.601,5.387,148.818
C03068=1222.766,-6.815,-41.295,-179.604,5.386,148.819
C03069=1222.771,-7.065,-41.281,-179.607,5.386,148.820
C03070=1222.777,-7.315,-41.267,-179.609,5.386,148.820
C03071=1222.782,-7.565,-41.253,-179.611,5.385,148.821
C03072=1222.787,-7.814,-41.239,-179.614,5.385,148.822
C03073=1222.792,-8.063,-41.225,-179.617,5.384,148.822
C03074=1222.796,-8.313,-41.211,-179.619,5.385,148.823
C03075=1222.801,-8.562,-41.197,-179.621,5.384,148.824
C03076=1222.807,-8.811,-41.183,-179.624,5.384,148.825
C03077=1222.812,-9.061,-41.169,-179.626,5.384,148.825
C03078=1222.817,-9.311,-41.155,-179.629,5.384,148.826
C03079=1222.823,-9.560,-41.141,-179.631,5.383,148.827
C03080=1222.828,-9.810,-41.127,-179.634,5.383,148.827
C03081=1222.832,-10.060,-41.113,-179.636,5.383,148.828
C03082=1222.837,-10.309,-41.099,-179.639,5.382,148.829
C03083=1222.843,-10.559,-41.086,-179.641,5.382,148.829
C03084=1222.848,-10.809,-41.072,-179.643,5.382,148.830
C03085=1222.852,-11.058,-41.057,-179.646,5.382,148.831
C03086=1222.857,-11.307,-41.044,-179.649,5.381,148.831
C03087=1222.862,-11.557,-41.030,-179.651,5.381,148.832
C03088=1222.868,-11.807,-41.016,-179.654,5.381,148.833
C03089=1222.873,-12.056,-41.002,-179.656,5.380,148.834
C03090=1222.877,-12.306,-40.989,-179.659,5.380,148.834
C03091=1222.882,-12.555,-40.974,-179.661,5.380,148.835
C03092=1222.888,-12.805,-40.961,-179.664,5.380,148.836
C03093=1222.893,-13.055,-40.947,-179.666,5.379,148.836
C03094=1222.897,-13.304,-40.933,-179.669,5.379,148.837
C03095=1222.903,-13.554,-40.920,-179.671,5.379,148.838
C03096=1222.908,-13.803,-40.906,-179.674,5.378,148.838
C03097=1222.913,-14.053,-40.891,-179.676,5.378,148.839
C03098=1222.918,-14.302,-40.878,-179.678,5.378,148.840
C03099=1222.923,-14.552,-40.865,-179.681,5.378,148.840
C03100=1222.929,-14.801,-40.851,-179.684,5.377,148.841
C03101=1222.934,-15.051,-40.836,-179.686,5.377,148.842
C03102=1222.938,-15.301,-40.823,-179.688,5.377,148.843
C03103=1222.944,-15.550,-40.809,-179.691,5.377,148.843
C03104=1222.949,-15.799,-40.795,-179.694,5.376,148.844
C03105=1222.953,-16.050,-40.782,-179.696,5.376,148.845
C03106=1222.959,-16.299,-40.768,-179.698,5.376,148.845
C03107=1222.964,-16.549,-40.755,-179.701,5.375,148.846
C03108=1222.969,-16.798,-40.741,-179.703,5.376,148.847
C03109=1222.974,-17.047,-40.727,-179.706,5.375,148.847
C03110=1222.979,-17.298,-40.714,-179.709,5.375,148.848
C03111=1222.984,-17.546,-40.700,-179.711,5.374,148.849
C03112=1222.989,-17.797,-40.687,-179.713,5.374,148.850
C03113=1222.995,-18.046,-40.673,-179.716,5.374,148.850
C03114=1222.999,-18.296,-40.660,-179.719,5.373,148.851
C03115=1223.004,-18.545,-40.646,-179.721,5.374,148.852
C03116=1223.010,-18.794,-40.632,-179.723,5.373,148.852
C03117=1223.014,-19.044,-40.619,-179.726,5.373,148.853
C03118=1223.020,-19.293,-40.605,-179.728,5.373,148.854
C03119=1223.024,-19.543,-40.592,-179.731,5.373,148.854
C03120=1223.030,-19.792,-40.578,-179.733,5.372,148.855
C03121=1223.035,-20.043,-40.564,-179.735,5.372,148.856
C03122=1223.040,-20.291,-40.551,-179.738,5.372,148.856
C03123=1223.045,-20.542,-40.537,-179.740,5.371,148.857
C03124=1223.049,-20.791,-40.524,-179.742,5.371,148.858
C03125=1223.055,-21.041,-40.511,-179.745,5.371,148.858
C03126=1223.060,-21.291,-40.496,-179.748,5.370,148.859
C03127=1223.065,-21.540,-40.484,-179.750,5.370,148.860
C03128=1223.070,-21.790,-40.469,-179.752,5.370,148.860
C03129=1223.075,-22.039,-40.457,-179.755,5.370,148.861
C03130=1223.081,-22.308,-40.442,-179.758,5.369,148.862
C03131=1223.087,-22.578,-40.428,-179.761,5.369,148.863
C03132=1223.093,-22.847,-40.413,-179.763,5.369,148.863
C03133=1223.097,-23.116,-40.399,-179.766,5.369,148.864
C03134=1223.103,-23.366,-40.385,-179.768,5.368,148.865
C03135=1223.108,-23.616,-40.372,-179.770,5.369,148.865
C03136=1223.113,-23.866,-40.358,-179.773,5.368,148.866
C03137=1223.118,-24.115,-40.346,-179.776,5.368,148.867
C03138=1223.123,-24.365,-40.331,-179.778,5.368,148.868
C03139=1223.128,-24.614,-40.319,-179.780,5.367,148.868
C03140=1223.133,-24.864,-40.305,-179.783,5.367,148.869
C03141=1223.138,-25.113,-40.292,-179.786,5.366,148.870
C03142=1223.143,-25.363,-40.278,-179.788,5.367,148.870
C03143=1223.148,-25.613,-40.266,-179.790,5.366,148.871
C03144=1223.153,-25.862,-40.251,-179.793,5.366,148.872
C03145=1223.158,-26.112,-40.239,-179.795,5.366,148.872
C03146=1223.164,-26.362,-40.225,-179.798,5.366,148.873
C03147=1223.168,-26.611,-40.212,-179.801,5.365,148.874
C03148=1223.174,-26.861,-40.198,-179.803,5.365,148.875
C03149=1223.179,-27.110,-40.186,-179.805,5.365,148.875
C03150=1223.184,-27.359,-40.172,-179.807,5.365,148.876
C03151=1223.189,-27.609,-40.159,-179.810,5.365,148.877
C03152=1223.194,-27.859,-40.146,-179.813,5.364,148.877
C03153=1223.199,-28.109,-40.133,-179.815,5.364,148.878
C03154=1223.204,-28.358,-40.119,-179.817,5.364,148.879
C03155=1223.209,-28.608,-40.106,-179.820,5.364,148.879
C03156=1223.215,-28.857,-40.093,-179.822,5.364,148.880
C03157=1223.219,-29.107,-40.080,-179.825,5.363,148.881
C03158=1223.225,-29.356,-40.066,-179.827,5.363,148.882
C03159=1223.230,-29.606,-40.054,-179.830,5.363,148.882
C03160=1223.235,-29.856,-40.040,-179.832,5.363,148.883
C03161=1223.240,-30.105,-40.028,-179.835,5.362,148.884
C03162=1223.244,-30.355,-40.014,-179.837,5.362,148.884
C03163=1223.250,-30.604,-40.001,-179.840,5.362,148.885
C03164=1223.255,-30.854,-39.988,-179.842,5.361,148.886
C03165=1223.261,-31.104,-39.974,-179.844,5.362,148.886
C03166=1223.266,-31.353,-39.962,-179.847,5.361,148.887
C03167=1223.270,-31.603,-39.949,-179.850,5.361,148.888
C03168=1223.276,-31.852,-39.935,-179.852,5.361,148.889
C03169=1223.281,-32.102,-39.922,-179.854,5.361,148.889
C03170=1223.285,-32.352,-39.909,-179.857,5.360,148.890
C03171=1223.291,-32.601,-39.896,-179.859,5.360,148.891
C03172=1223.296,-32.851,-39.883,-179.862,5.360,148.891
C03173=1223.301,-33.101,-39.871,-179.865,5.359,148.892
C03174=1223.307,-33.350,-39.857,-179.867,5.360,148.893
C03175=1223.311,-33.600,-39.844,-179.869,5.359,148.893
C03176=1223.316,-33.849,-39.831,-179.871,5.360,148.894
C03177=1223.322,-34.099,-39.818,-179.874,5.359,148.895
C03178=1223.327,-34.349,-39.805,-179.877,5.359,148.895
C03179=1223.332,-34.598,-39.792,-179.879,5.359,148.896
C03180=1223.336,-34.848,-39.779,-179.881,5.358,148.897
C03181=1223.342,-35.098,-39.766,-179.884,5.358,148.898
C03182=1223.347,-35.347,-39.754,-179.886,5.358,148.898
C03183=1223.352,-35.597,-39.741,-179.889,5.358,148.899
C03184=1223.358,-35.846,-39.727,-179.891,5.357,148.900
C03185=1223.363,-36.096,-39.715,-179.894,5.358,148.900
C03186=1223.367,-36.346,-39.702,-179.896,5.357,148.901
C03187=1223.372,-36.595,-39.689,-179.898,5.358,148.902
C03188=1223.378,-36.845,-39.676,-179.901,5.357,148.902
C03189=1223.383,-37.095,-39.663,-179.904,5.357,148.903
C03190=1223.388,-37.344,-39.651,-179.906,5.357,148.904
C03191=1223.393,-37.593,-39.638,-179.908,5.356,148.905
C03192=1223.399,-37.843,-39.625,-179.911,5.356,148.905
C03193=1223.403,-38.093,-39.612,-179.913,5.356,148.906
C03194=1223.408,-38.342,-39.599,-179.916,5.356,148.907
C03195=1223.414,-38.592,-39.587,-179.918,5.356,148.907
C03196=1223.418,-38.842,-39.574,-179.921,5.356,148.908
C03197=1223.424,-39.091,-39.560,-179.923,5.355,148.909
C03198=1223.429,-39.341,-39.548,-179.925,5.355,148.909
C03199=1223.434,-39.590,-39.535,-179.928,5.355,148.910
C03200=1223.439,-39.840,-39.522,-179.931,5.354,148.911
C03201=1223.444,-40.089,-39.510,-179.933,5.355,148.912
C03202=1223.450,-40.340,-39.497,-179.935,5.354,148.912
C03203=1223.455,-40.590,-39.484,-179.937,5.355,148.913
C03204=1223.460,-40.839,-39.472,-179.940,5.354,148.914
C03205=1223.465,-41.088,-39.459,-179.943,5.354,148.914
C03206=1223.470,-41.338,-39.446,-179.945,5.354,148.915
C03207=1223.474,-41.588,-39.433,-179.948,5.353,148.916
C03208=1223.480,-41.837,-39.421,-179.950,5.353,148.916
C03209=1223.485,-42.086,-39.408,-179.952,5.353,148.917
C03210=1223.491,-42.336,-39.396,-179.955,5.353,148.918
C03211=1223.495,-42.586,-39.383,-179.957,5.353,148.919
C03212=1223.501,-42.836,-39.370,-179.960,5.353,148.919
C03213=1223.506,-43.085,-39.358,-179.962,5.352,148.920
C03214=1223.511,-43.334,-39.345,-179.964,5.353,148.921
C03215=1223.515,-43.584,-39.332,-179.967,5.352,148.921
C03216=1223.521,-43.834,-39.320,-179.969,5.352,148.922
C03217=1223.526,-44.084,-39.308,-179.972,5.352,148.923
C03218=1223.532,-44.333,-39.294,-179.974,5.351,148.924
C03219=1223.537,-44.583,-39.282,-179.977,5.352,148.924
C03220=1223.541,-44.833,-39.269,-179.979,5.351,148.925
C03221=1223.547,-45.083,-39.257,-179.982,5.351,148.926
C03222=1223.552,-45.332,-39.244,-179.984,5.351,148.926
C03223=1223.557,-45.581,-39.232,-179.987,5.351,148.927
C03224=1223.562,-45.831,-39.219,-179.989,5.351,148.928
C03225=1223.567,-46.081,-39.207,-179.991,5.350,148.928
C03226=1223.572,-46.330,-39.194,-179.994,5.350,148.929
C03227=1223.577,-46.580,-39.182,-179.996,5.350,148.930
C03228=1223.583,-46.830,-39.170,-179.999,5.350,148.931
C03229=1223.588,-47.079,-39.157,179.999,5.350,148.931
C03230=1223.592,-47.329,-39.144,179.996,5.350,148.932
C03231=1223.597,-47.578,-39.132,179.994,5.349,148.933
C03232=1223.603,-47.828,-39.120,179.992,5.350,148.933
C03233=1223.608,-48.078,-39.107,179.989,5.349,148.934
C03234=1223.614,-48.348,-39.094,179.986,5.349,148.935
C03235=1223.620,-48.617,-39.080,179.984,5.349,148.935
C03236=1223.625,-48.887,-39.067,179.982,5.348,148.936
C03237=1223.630,-49.157,-39.054,179.978,5.348,148.937
C03238=1223.635,-49.407,-39.041,179.976,5.349,148.938
C03239=1223.640,-49.657,-39.029,179.974,5.348,148.938
C03240=1223.646,-49.906,-39.016,179.972,5.348,148.939
C03241=1223.651,-50.155,-39.004,179.969,5.348,148.940
C03242=1223.656,-50.405,-38.992,179.967,5.347,148.940
C03243=1223.661,-50.655,-38.979,179.965,5.348,148.941
C03244=1223.666,-50.905,-38.966,179.962,5.347,148.942
C03245=1223.671,-51.155,-38.955,179.960,5.347,148.942
C03246=1223.676,-51.404,-38.942,179.957,5.347,148.943
C03247=1223.682,-51.654,-38.930,179.955,5.346,148.944
C03248=1223.687,-51.903,-38.917,179.953,5.347,148.945
C03249=1223.692,-52.153,-38.906,179.950,5.346,148.945
C03250=1223.697,-52.402,-38.893,179.948,5.347,148.946
C03251=1223.702,-52.653,-38.881,179.945,5.346,148.947
C03252=1223.707,-52.902,-38.868,179.942,5.346,148.947
C03253=1223.712,-53.151,-38.856,179.940,5.346,148.948
C03254=1223.717,-53.401,-38.844,179.938,5.346,148.949
C03255=1223.722,-53.651,-38.832,179.936,5.346,148.950
C03256=1223.728,-53.901,-38.820,179.933,5.345,148.950
C03257=1223.733,-54.150,-38.807,179.931,5.346,148.951
C03258=1223.738,-54.400,-38.795,179.928,5.345,148.952
C03259=1223.743,-54.649,-38.783,179.925,5.345,148.952
C03260=1223.749,-54.899,-38.771,179.923,5.345,148.953
C03261=1223.753,-55.148,-38.759,179.921,5.345,148.954
C03262=1223.758,-55.399,-38.747,179.919,5.345,148.954
C03263=1223.763,-55.648,-38.734,179.916,5.344,148.955
C03264=1223.769,-55.898,-38.722,179.913,5.344,148.956
C03265=1223.774,-56.148,-38.710,179.911,5.344,148.957
C03266=1223.779,-56.397,-38.698,179.909,5.344,148.957
C03267=1223.784,-56.647,-38.686,179.906,5.344,148.958
C03268=1223.789,-56.896,-38.674,179.904,5.344,148.959
C03269=1223.794,-57.146,-38.662,179.902,5.344,148.959
C03270=1223.800,-57.395,-38.649,179.899,5.344,148.960
C03271=1223.805,-57.645,-38.637,179.896,5.343,148.961
C03272=1223.810,-57.895,-38.625,179.894,5.343,148.961
C03273=1223.815,-58.144,-38.613,179.892,5.343,148.962
C03274=1223.820,-58.394,-38.602,179.890,5.343,148.963
C03275=1223.826,-58.644,-38.590,179.887,5.343,148.964
C03276=1223.831,-58.893,-38.577,179.885,5.343,148.964
C03277=1223.836,-59.143,-38.566,179.882,5.343,148.965
C03278=1223.841,-59.392,-38.553,179.879,5.342,148.966
C03279=1223.846,-59.642,-38.541,179.877,5.343,148.966
C03280=1223.851,-59.892,-38.529,179.875,5.342,148.967
C03281=1223.856,-60.141,-38.517,179.873,5.342,148.968
C03282=1223.861,-60.391,-38.505,179.870,5.342,148.969
C03283=1223.867,-60.641,-38.494,179.868,5.342,148.969
C03284=1223.872,-60.890,-38.481,179.865,5.342,148.970
C03285=1223.877,-61.140,-38.470,179.863,5.341,148.971
C03286=1223.882,-61.390,-38.458,179.860,5.342,148.971
C03287=1223.887,-61.640,-38.446,179.858,5.341,148.972
C03288=1223.893,-61.889,-38.433,179.856,5.342,148.973
C03289=1223.897,-62.139,-38.422,179.853,5.341,148.973
C03290=1223.903,-62.389,-38.410,179.851,5.342,148.974
C03291=1223.908,-62.638,-38.398,179.848,5.341,148.975
C03292=1223.912,-62.888,-38.386,179.846,5.341,148.976
C03293=1223.918,-63.138,-38.374,179.844,5.341,148.976
C03294=1223.923,-63.388,-38.362,179.841,5.340,148.977
C03295=1223.929,-63.638,-38.351,179.839,5.341,148.978
C03296=1223.933,-63.887,-38.339,179.836,5.340,148.978
C03297=1223.939,-64.137,-38.327,179.834,5.341,148.979
C03298=1223.944,-64.386,-38.315,179.832,5.340,148.980
C03299=1223.949,-64.636,-38.304,179.830,5.340,148.980
C03300=1223.954,-64.885,-38.291,179.827,5.340,148.981
C03301=1223.959,-65.135,-38.279,179.824,5.339,148.982
C03302=1223.964,-65.385,-38.268,179.822,5.340,148.982
C03303=1223.970,-65.634,-38.256,179.820,5.339,148.983
C03304=1223.975,-65.884,-38.244,179.818,5.339,148.984
C03305=1223.980,-66.134,-38.233,179.815,5.339,148.985
C03306=1223.985,-66.383,-38.220,179.813,5.339,148.985
C03307=1223.990,-66.633,-38.209,179.810,5.339,148.986
C03308=1223.995,-66.883,-38.197,179.808,5.339,148.987
C03309=1224.001,-67.133,-38.185,179.805,5.339,148.987
C03310=1224.005,-67.382,-38.174,179.803,5.339,148.988
C03311=1224.011,-67.632,-38.162,179.801,5.339,148.989
C03312=1224.016,-67.882,-38.150,179.798,5.338,148.989
C03313=1224.021,-68.132,-38.139,179.796,5.339,148.990
C03314=1224.027,-68.380,-38.127,179.793,5.338,148.991
C03315=1224.031,-68.630,-38.116,179.791,5.338,148.992
C03316=1224.037,-68.880,-38.104,179.788,5.338,148.992
C03317=1224.042,-69.129,-38.092,179.786,5.338,148.993
C03318=1224.047,-69.379,-38.080,179.784,5.338,148.994
C03319=1224.052,-69.629,-38.069,179.782,5.338,148.994
C03320=1224.057,-69.879,-38.057,179.779,5.338,148.995
C03321=1224.063,-70.129,-38.045,179.776,5.337,148.996
C03322=1224.068,-70.378,-38.034,179.774,5.338,148.997
C03323=1224.073,-70.628,-38.023,179.771,5.337,148.997
C03324=1224.078,-70.877,-38.011,179.769,5.338,148.998
C03325=1224.083,-71.127,-37.999,179.767,5.337,148.999
C03326=1224.089,-71.377,-37.988,179.765,5.337,148.999
C03327=1224.093,-71.627,-37.976,179.762,5.337,149.000
C03328=1224.100,-71.876,-37.965,179.760,5.337,149.001
C03329=1224.104,-72.126,-37.953,179.757,5.337,149.002
C03330=1224.110,-72.376,-37.942,179.755,5.337,149.002
C03331=1224.114,-72.625,-37.930,179.753,5.336,149.003
C03332=1224.120,-72.875,-37.918,179.751,5.337,149.003
C03333=1224.124,-73.125,-37.907,179.748,5.336,149.004
C03334=1224.130,-73.374,-37.896,179.746,5.336,149.005
C03335=1224.135,-73.624,-37.884,179.743,5.336,149.006
C03336=1224.141,-73.874,-37.872,179.741,5.336,149.006
C03337=1224.145,-74.123,-37.861,179.739,5.336,149.007
C03338=1224.151,-74.394,-37.849,179.736,5.336,149.008
C03339=1224.157,-74.664,-37.836,179.733,5.336,149.009
C03340=1224.162,-74.935,-37.824,179.731,5.336,149.009
C03341=1224.168,-75.205,-37.811,179.728,5.335,149.010
C03342=1224.173,-75.455,-37.801,179.726,5.336,149.011
C03343=1224.179,-75.705,-37.789,179.723,5.335,149.011
C03344=1224.183,-75.954,-37.778,179.721,5.336,149.012
C03345=1224.189,-76.204,-37.766,179.719,5.335,149.013
C03346=1224.194,-76.453,-37.755,179.716,5.336,149.014
C03347=1224.199,-76.703,-37.744,179.714,5.335,149.014
C03348=1224.204,-76.953,-37.732,179.712,5.335,149.015
C03349=1224.209,-77.202,-37.720,179.709,5.335,149.016
C03350=1224.215,-77.452,-37.710,179.706,5.334,149.016
C03351=1224.220,-77.702,-37.698,179.704,5.335,149.017
C03352=1224.225,-77.952,-37.687,179.702,5.334,149.018
C03353=1224.230,-78.201,-37.675,179.700,5.335,149.019
C03354=1224.235,-78.450,-37.664,179.697,5.334,149.019
C03355=1224.241,-78.701,-37.653,179.695,5.334,149.020
C03356=1224.246,-78.951,-37.642,179.693,5.334,149.020
C03357=1224.251,-79.200,-37.630,179.690,5.334,149.021
C03358=1224.257,-79.449,-37.619,179.688,5.334,149.022
C03359=1224.261,-79.699,-37.608,179.686,5.334,149.023
C03360=1224.266,-79.949,-37.597,179.683,5.334,149.023
C03361=1224.272,-80.199,-37.585,179.681,5.334,149.024
C03362=1224.277,-80.448,-37.574,179.678,5.334,149.025
C03363=1224.282,-80.698,-37.562,179.676,5.334,149.025
C03364=1224.287,-80.948,-37.552,179.674,5.333,149.026
C03365=1224.293,-81.197,-37.541,179.671,5.334,149.027
C03366=1224.298,-81.447,-37.529,179.669,5.333,149.028
C03367=1224.303,-81.697,-37.518,179.667,5.334,149.028
C03368=1224.308,-81.947,-37.507,179.664,5.333,149.029
C03369=1224.314,-82.196,-37.496,179.662,5.334,149.030
C03370=1224.319,-82.446,-37.484,179.659,5.333,149.030
C03371=1224.324,-82.696,-37.474,179.657,5.333,149.031
C03372=1224.329,-82.945,-37.463,179.654,5.333,149.032
C03373=1224.334,-83.195,-37.451,179.652,5.332,149.032
C03374=1224.339,-83.445,-37.440,179.650,5.333,149.033
C03375=1224.344,-83.695,-37.429,179.648,5.332,149.034
C03376=1224.350,-83.944,-37.418,179.645,5.332,149.034
C03377=1224.355,-84.194,-37.407,179.643,5.332,149.035
C03378=1224.360,-84.444,-37.396,179.641,5.332,149.036
C03379=1224.365,-84.693,-37.385,179.638,5.332,149.037
C03380=1224.371,-84.944,-37.374,179.636,5.332,149.037
C03381=1224.375,-85.193,-37.362,179.633,5.332,149.038
C03382=1224.381,-85.442,-37.351,179.631,5.332,149.039
C03383=1224.386,-85.692,-37.341,179.628,5.332,149.039
C03384=1224.391,-85.942,-37.329,179.626,5.332,149.040
C03385=1224.397,-86.192,-37.319,179.624,5.332,149.041
C03386=1224.401,-86.441,-37.307,179.622,5.332,149.041
C03387=1224.406,-86.691,-37.296,179.619,5.332,149.042
C03388=1224.412,-86.941,-37.286,179.617,5.332,149.043
C03389=1224.417,-87.191,-37.274,179.614,5.331,149.044
C03390=1224.423,-87.440,-37.264,179.613,5.331,149.044
C03391=1224.427,-87.690,-37.253,179.610,5.331,149.045
C03392=1224.432,-87.940,-37.242,179.608,5.331,149.046
C03393=1224.438,-88.189,-37.231,179.605,5.331,149.046
C03394=1224.443,-88.439,-37.219,179.603,5.331,149.047
C03395=1224.448,-88.689,-37.209,179.600,5.331,149.048
C03396=1224.453,-88.938,-37.198,179.598,5.331,149.048
C03397=1224.458,-89.188,-37.187,179.596,5.331,149.049
C03398=1224.464,-89.437,-37.176,179.594,5.331,149.050
C03399=1224.469,-89.687,-37.166,179.591,5.331,149.050
C03400=1224.474,-89.937,-37.154,179.589,5.331,149.051
C03401=1224.480,-90.187,-37.143,179.586,5.331,149.052
C03402=1224.484,-90.436,-37.132,179.584,5.331,149.053
C03403=1224.490,-90.686,-37.122,179.581,5.330,149.053
C03404=1224.495,-90.936,-37.111,179.580,5.330,149.054
C03405=1224.500,-91.186,-37.100,179.577,5.330,149.055
C03406=1224.506,-91.436,-37.089,179.575,5.330,149.055
C03407=1224.511,-91.685,-37.078,179.572,5.330,149.056
C03408=1224.516,-91.935,-37.068,179.570,5.330,149.057
C03409=1224.521,-92.185,-37.057,179.568,5.330,149.057
C03410=1224.527,-92.434,-37.046,179.565,5.330,149.058
C03411=1224.531,-92.684,-37.035,179.563,5.330,149.059
C03412=1224.536,-92.934,-37.024,179.561,5.330,149.060
C03413=1224.542,-93.184,-37.014,179.558,5.330,149.060
C03414=1224.547,-93.433,-37.003,179.556,5.330,149.061
C03415=1224.552,-93.683,-36.993,179.553,5.330,149.062
C03416=1224.558,-93.933,-36.981,179.552,5.330,149.062
C03417=1224.563,-94.182,-36.971,179.549,5.329,149.063
C03418=1224.568,-94.432,-36.960,179.547,5.330,149.064
C03419=1224.574,-94.681,-36.949,179.544,5.329,149.064
C03420=1224.579,-94.932,-36.939,179.542,5.329,149.065
C03421=1224.584,-95.181,-36.928,179.539,5.329,149.066
C03422=1224.589,-95.431,-36.917,179.537,5.329,149.066
C03423=1224.594,-95.681,-36.906,179.535,5.329,149.067
C03424=1224.599,-95.931,-36.896,179.533,5.329,149.068
C03425=1224.604,-96.180,-36.885,179.530,5.329,149.069
C03426=1224.610,-96.430,-36.875,179.528,5.329,149.069
C03427=1224.615,-96.680,-36.864,179.525,5.329,149.070
C03428=1224.620,-96.929,-36.853,179.524,5.329,149.070
C03429=1224.625,-97.179,-36.843,179.521,5.328,149.071
C03430=1224.631,-97.429,-36.833,179.519,5.329,149.072
C03431=1224.635,-97.678,-36.821,179.516,5.328,149.073
C03432=1224.641,-97.928,-36.811,179.514,5.329,149.073
C03433=1224.646,-98.178,-36.800,179.511,5.328,149.074
C03434=1224.652,-98.428,-36.790,179.509,5.329,149.075
C03435=1224.656,-98.677,-36.779,179.507,5.329,149.075
C03436=1224.662,-98.927,-36.769,179.504,5.328,149.076
C03437=1224.667,-99.176,-36.759,179.502,5.329,149.077
C03438=1224.672,-99.427,-36.748,179.500,5.328,149.078
C03439=1224.678,-99.675,-36.737,179.498,5.328,149.078
C03440=1224.683,-99.926,-36.726,179.495,5.328,149.079
C03441=1224.688,-100.175,-36.716,179.493,5.328,149.079
C03442=1224.694,-100.447,-36.705,179.491,5.328,149.080
C03443=1224.699,-100.718,-36.693,179.488,5.327,149.081
C03444=1224.706,-100.988,-36.682,179.485,5.328,149.082
C03445=1224.711,-101.260,-36.671,179.483,5.328,149.083
C03446=1224.715,-101.509,-36.660,179.481,5.328,149.083
C03447=1224.721,-101.759,-36.649,179.478,5.328,149.084
C03448=1224.726,-102.009,-36.639,179.476,5.328,149.084
C03449=1224.732,-102.259,-36.629,179.474,5.327,149.085
C03450=1224.737,-102.508,-36.618,179.472,5.328,149.086
C03451=1224.742,-102.759,-36.608,179.469,5.327,149.087
C03452=1224.748,-103.007,-36.597,179.467,5.328,149.087
C03453=1224.752,-103.257,-36.587,179.464,5.327,149.088
C03454=1224.757,-103.507,-36.577,179.462,5.327,149.089
C03455=1224.762,-103.757,-36.566,179.459,5.327,149.089
C03456=1224.768,-104.007,-36.556,179.457,5.327,149.090
C03457=1224.774,-104.256,-36.546,179.455,5.327,149.091
C03458=1224.779,-104.506,-36.535,179.453,5.327,149.091
C03459=1224.784,-104.756,-36.525,179.450,5.327,149.092
C03460=1224.789,-105.006,-36.514,179.448,5.327,149.093
C03461=1224.794,-105.256,-36.505,179.446,5.327,149.094
C03462=1224.799,-105.504,-36.494,179.443,5.327,149.094
C03463=1224.804,-105.755,-36.483,179.441,5.327,149.095
C03464=1224.810,-106.004,-36.473,179.439,5.327,149.096
C03465=1224.815,-106.254,-36.463,179.437,5.327,149.096
C03466=1224.821,-106.504,-36.452,179.434,5.326,149.097
C03467=1224.825,-106.753,-36.443,179.432,5.327,149.098
C03468=1224.830,-107.003,-36.432,179.430,5.326,149.098
C03469=1224.836,-107.253,-36.422,179.428,5.327,149.099
C03470=1224.842,-107.503,-36.412,179.425,5.326,149.100
C03471=1224.847,-107.753,-36.401,179.423,5.327,149.100
C03472=1224.852,-108.002,-36.391,179.420,5.326,149.101
C03473=1224.856,-108.252,-36.381,179.418,5.327,149.102
C03474=1224.862,-108.502,-36.371,179.416,5.326,149.102
C03475=1224.868,-108.751,-36.361,179.414,5.326,149.103
C03476=1224.873,-109.002,-36.350,179.411,5.326,149.104
C03477=1224.878,-109.251,-36.340,179.409,5.326,149.105
C03478=1224.883,-109.500,-36.330,179.407,5.326,149.105
C03479=1224.888,-109.751,-36.320,179.404,5.326,149.106
C03480=1224.894,-110.000,-36.309,179.402,5.326,149.107
C03481=1224.899,-110.250,-36.299,179.399,5.326,149.107
C03482=1224.904,-110.500,-36.289,179.398,5.326,149.108
C03483=1224.909,-110.749,-36.279,179.395,5.325,149.109
C03484=1224.915,-110.999,-36.269,179.393,5.326,149.109
C03485=1224.920,-111.250,-36.259,179.390,5.325,149.110
C03486=1224.925,-111.499,-36.249,179.388,5.326,149.111
C03487=1224.931,-111.748,-36.239,179.386,5.325,149.111
C03488=1224.936,-111.999,-36.228,179.384,5.326,149.112
C03489=1224.941,-112.248,-36.218,179.381,5.325,149.113
C03490=1224.946,-112.497,-36.209,179.379,5.325,149.113
C03491=1224.952,-112.747,-36.198,179.377,5.325,149.114
C03492=1224.957,-112.997,-36.188,179.374,5.325,149.115
C03493=1224.962,-113.247,-36.179,179.372,5.326,149.115
C03494=1224.967,-113.497,-36.169,179.370,5.325,149.116
C03495=1224.972,-113.747,-36.158,179.368,5.326,149.117
C03496=1224.978,-113.996,-36.148,179.365,5.325,149.117
C03497=1224.983,-114.246,-36.138,179.363,5.325,149.118
C03498=1224.988,-114.495,-36.128,179.361,5.325,149.119
C03499=1224.994,-114.746,-36.118,179.359,5.325,149.120
C03500=1224.999,-114.995,-36.109,179.356,5.325,149.120
C03501=1225.004,-115.245,-36.098,179.354,5.325,149.121
C03502=1225.009,-115.495,-36.088,179.351,5.325,149.122
C03503=1225.014,-115.744,-36.078,179.349,5.325,149.122
C03504=1225.020,-115.994,-36.069,179.347,5.324,149.123
C03505=1225.026,-116.244,-36.059,179.345,5.325,149.124
C03506=1225.030,-116.494,-36.049,179.343,5.325,149.124
C03507=1225.035,-116.743,-36.038,179.340,5.325,149.125
C03508=1225.040,-116.993,-36.029,179.338,5.325,149.126
C03509=1225.046,-117.243,-36.019,179.335,5.325,149.126
C03510=1225.051,-117.493,-36.009,179.334,5.324,149.127
C03511=1225.056,-117.742,-35.999,179.331,5.324,149.128
C03512=1225.062,-117.992,-35.989,179.329,5.324,149.128
C03513=1225.068,-118.242,-35.979,179.326,5.324,149.129
C03514=1225.072,-118.492,-35.969,179.324,5.324,149.130
C03515=1225.077,-118.742,-35.959,179.321,5.324,149.131
C03516=1225.083,-118.991,-35.950,179.320,5.324,149.131
C03517=1225.088,-119.241,-35.940,179.318,5.324,149.132
C03518=1225.094,-119.490,-35.930,179.315,5.324,149.132
C03519=1225.098,-119.740,-35.920,179.313,5.324,149.133
C03520=1225.104,-119.991,-35.910,179.310,5.324,149.134
C03521=1225.109,-120.240,-35.901,179.308,5.324,149.135
C03522=1225.114,-120.489,-35.891,179.306,5.323,149.135
C03523=1225.120,-120.739,-35.882,179.304,5.324,149.136
C03524=1225.125,-120.989,-35.871,179.301,5.323,149.137
C03525=1225.129,-121.239,-35.862,179.299,5.324,149.137
C03526=1225.135,-121.489,-35.852,179.296,5.323,149.138
C03527=1225.141,-121.738,-35.842,179.294,5.324,149.139
C03528=1225.146,-121.988,-35.833,179.293,5.324,149.139
C03529=1225.151,-122.238,-35.822,179.290,5.323,149.140
C03530=1225.156,-122.488,-35.813,179.288,5.324,149.141
C03531=1225.162,-122.738,-35.803,179.285,5.323,149.141
C03532=1225.167,-122.987,-35.794,179.283,5.324,149.142
C03533=1225.172,-123.237,-35.783,179.281,5.323,149.143
C03534=1225.177,-123.486,-35.775,179.279,5.323,149.143
C03535=1225.182,-123.737,-35.764,179.276,5.323,149.144
C03536=1225.188,-123.987,-35.755,179.274,5.323,149.145
C03537=1225.193,-124.236,-35.745,179.272,5.324,149.145
C03538=1225.198,-124.486,-35.736,179.269,5.323,149.146
C03539=1225.204,-124.735,-35.726,179.268,5.323,149.147
C03540=1225.209,-124.985,-35.716,179.265,5.323,149.147
C03541=1225.215,-125.235,-35.707,179.263,5.323,149.148
C03542=1225.219,-125.485,-35.697,179.260,5.323,149.149
C03543=1225.225,-125.735,-35.687,179.258,5.323,149.149
C03544=1225.230,-125.984,-35.678,179.256,5.322,149.150
C03545=1225.235,-126.234,-35.669,179.254,5.323,149.151
C03546=1224.814,-126.245,-35.704,179.249,5.326,149.153
C03547=1224.808,-125.995,-35.714,179.251,5.326,149.152
C03548=1224.803,-125.746,-35.724,179.254,5.326,149.151
C03549=1224.797,-125.496,-35.733,179.256,5.326,149.151
C03550=1224.793,-125.246,-35.743,179.258,5.327,149.150
C03551=1224.787,-124.995,-35.752,179.261,5.326,149.149
C03552=1224.782,-124.746,-35.762,179.263,5.327,149.149
C03553=1224.776,-124.496,-35.772,179.265,5.326,149.148
C03554=1224.771,-124.247,-35.781,179.267,5.326,149.147
C03555=1224.766,-123.997,-35.791,179.270,5.326,149.147
C03556=1224.761,-123.747,-35.800,179.272,5.326,149.146
C03557=1224.756,-123.497,-35.811,179.274,5.327,149.145
C03558=1224.751,-123.247,-35.820,179.276,5.326,149.145
C03559=1224.745,-122.998,-35.830,179.279,5.327,149.144
C03560=1224.740,-122.748,-35.839,179.281,5.326,149.143
C03561=1224.734,-122.498,-35.849,179.283,5.327,149.143
C03562=1224.729,-122.249,-35.859,179.286,5.327,149.142
C03563=1224.724,-121.998,-35.869,179.288,5.327,149.141
C03564=1224.719,-121.749,-35.878,179.290,5.327,149.141
C03565=1224.714,-121.500,-35.888,179.292,5.327,149.140
C03566=1224.708,-121.250,-35.897,179.295,5.327,149.139
C03567=1224.703,-121.000,-35.907,179.297,5.327,149.139
C03568=1224.698,-120.750,-35.917,179.299,5.327,149.138
C03569=1224.693,-120.500,-35.927,179.301,5.327,149.137
C03570=1224.688,-120.251,-35.937,179.304,5.327,149.136
C03571=1224.682,-120.001,-35.946,179.306,5.327,149.136
C03572=1224.676,-119.751,-35.956,179.308,5.328,149.135
C03573=1224.672,-119.501,-35.966,179.311,5.327,149.135
C03574=1224.666,-119.252,-35.976,179.313,5.328,149.134
C03575=1224.661,-119.002,-35.985,179.315,5.328,149.133
C03576=1224.656,-118.752,-35.996,179.317,5.327,149.132
C03577=1224.651,-118.503,-36.005,179.320,5.328,149.132
C03578=1224.645,-118.252,-36.015,179.322,5.328,149.131
C03579=1224.640,-118.003,-36.025,179.324,5.328,149.130
C03580=1224.635,-117.753,-36.035,179.326,5.328,149.130
C03581=1224.629,-117.504,-36.045,179.329,5.328,149.129
C03582=1224.624,-117.253,-36.055,179.331,5.328,149.128
C03583=1224.619,-117.004,-36.065,179.334,5.328,149.128
C03584=1224.614,-116.754,-36.075,179.336,5.328,149.127
C03585=1224.609,-116.505,-36.084,179.338,5.328,149.126
C03586=1224.603,-116.254,-36.094,179.340,5.328,149.126
C03587=1224.598,-116.005,-36.104,179.342,5.328,149.125
C03588=1224.593,-115.755,-36.114,179.345,5.328,149.124
C03589=1224.587,-115.506,-36.124,179.347,5.328,149.124
C03590=1224.582,-115.256,-36.135,179.350,5.328,149.123
C03591=1224.577,-115.006,-36.144,179.351,5.328,149.122
C03592=1224.572,-114.756,-36.154,179.354,5.329,149.122
C03593=1224.566,-114.507,-36.164,179.356,5.328,149.121
C03594=1224.562,-114.257,-36.174,179.359,5.329,149.120
C03595=1224.556,-114.007,-36.184,179.361,5.328,149.120
C03596=1224.550,-113.757,-36.194,179.364,5.329,149.119
C03597=1224.545,-113.508,-36.203,179.366,5.328,149.118
C03598=1224.540,-113.257,-36.214,179.368,5.329,149.118
C03599=1224.535,-113.008,-36.224,179.370,5.329,149.117
C03600=1224.529,-112.758,-36.234,179.372,5.328,149.116
C03601=1224.525,-112.508,-36.244,179.375,5.329,149.115
C03602=1224.519,-112.259,-36.255,179.377,5.328,149.115
C03603=1224.513,-112.009,-36.264,179.380,5.329,149.114
C03604=1224.509,-111.759,-36.274,179.382,5.329,149.113
C03605=1224.504,-111.509,-36.284,179.384,5.329,149.113
C03606=1224.498,-111.260,-36.295,179.386,5.329,149.112
C03607=1224.492,-111.010,-36.305,179.389,5.329,149.111
C03608=1224.488,-110.760,-36.315,179.391,5.329,149.111
C03609=1224.483,-110.511,-36.325,179.393,5.329,149.110
C03610=1224.477,-110.261,-36.335,179.395,5.329,149.109
C03611=1224.472,-110.011,-36.346,179.398,5.329,149.109
C03612=1224.467,-109.762,-36.355,179.400,5.330,149.108
C03613=1224.461,-109.512,-36.366,179.402,5.330,149.107
C03614=1224.456,-109.262,-36.376,179.404,5.330,149.107
C03615=1224.451,-109.012,-36.386,179.407,5.329,149.106
C03616=1224.445,-108.763,-36.397,179.409,5.330,149.105
C03617=1224.441,-108.513,-36.406,179.411,5.329,149.104
C03618=1224.435,-108.263,-36.417,179.414,5.330,149.104
C03619=1224.430,-108.013,-36.427,179.416,5.330,149.103
C03620=1224.425,-107.764,-36.437,179.418,5.330,149.103
C03621=1224.420,-107.514,-36.447,179.420,5.330,149.102
C03622=1224.415,-107.264,-36.458,179.423,5.330,149.101
C03623=1224.409,-107.015,-36.468,179.425,5.330,149.100
C03624=1224.404,-106.765,-36.478,179.428,5.330,149.100
C03625=1224.399,-106.515,-36.489,179.430,5.330,149.099
C03626=1224.393,-106.265,-36.499,179.433,5.330,149.098
C03627=1224.389,-106.015,-36.509,179.434,5.330,149.098
C03628=1224.383,-105.766,-36.519,179.437,5.331,149.097
C03629=1224.378,-105.516,-36.529,179.439,5.330,149.096
C03630=1224.373,-105.266,-36.540,179.442,5.331,149.096
C03631=1224.367,-105.016,-36.550,179.444,5.330,149.095
C03632=1224.362,-104.766,-36.561,179.446,5.330,149.094
C03633=1224.357,-104.517,-36.571,179.449,5.330,149.094
C03634=1224.352,-104.267,-36.580,179.451,5.330,149.093
C03635=1224.347,-104.017,-36.591,179.453,5.331,149.092
C03636=1224.341,-103.768,-36.601,179.455,5.331,149.092
C03637=1224.336,-103.518,-36.613,179.458,5.331,149.091
C03638=1224.331,-103.268,-36.623,179.460,5.331,149.090
C03639=1224.325,-103.019,-36.633,179.462,5.331,149.089
C03640=1224.320,-102.769,-36.644,179.464,5.331,149.089
C03641=1224.315,-102.519,-36.654,179.467,5.331,149.088
